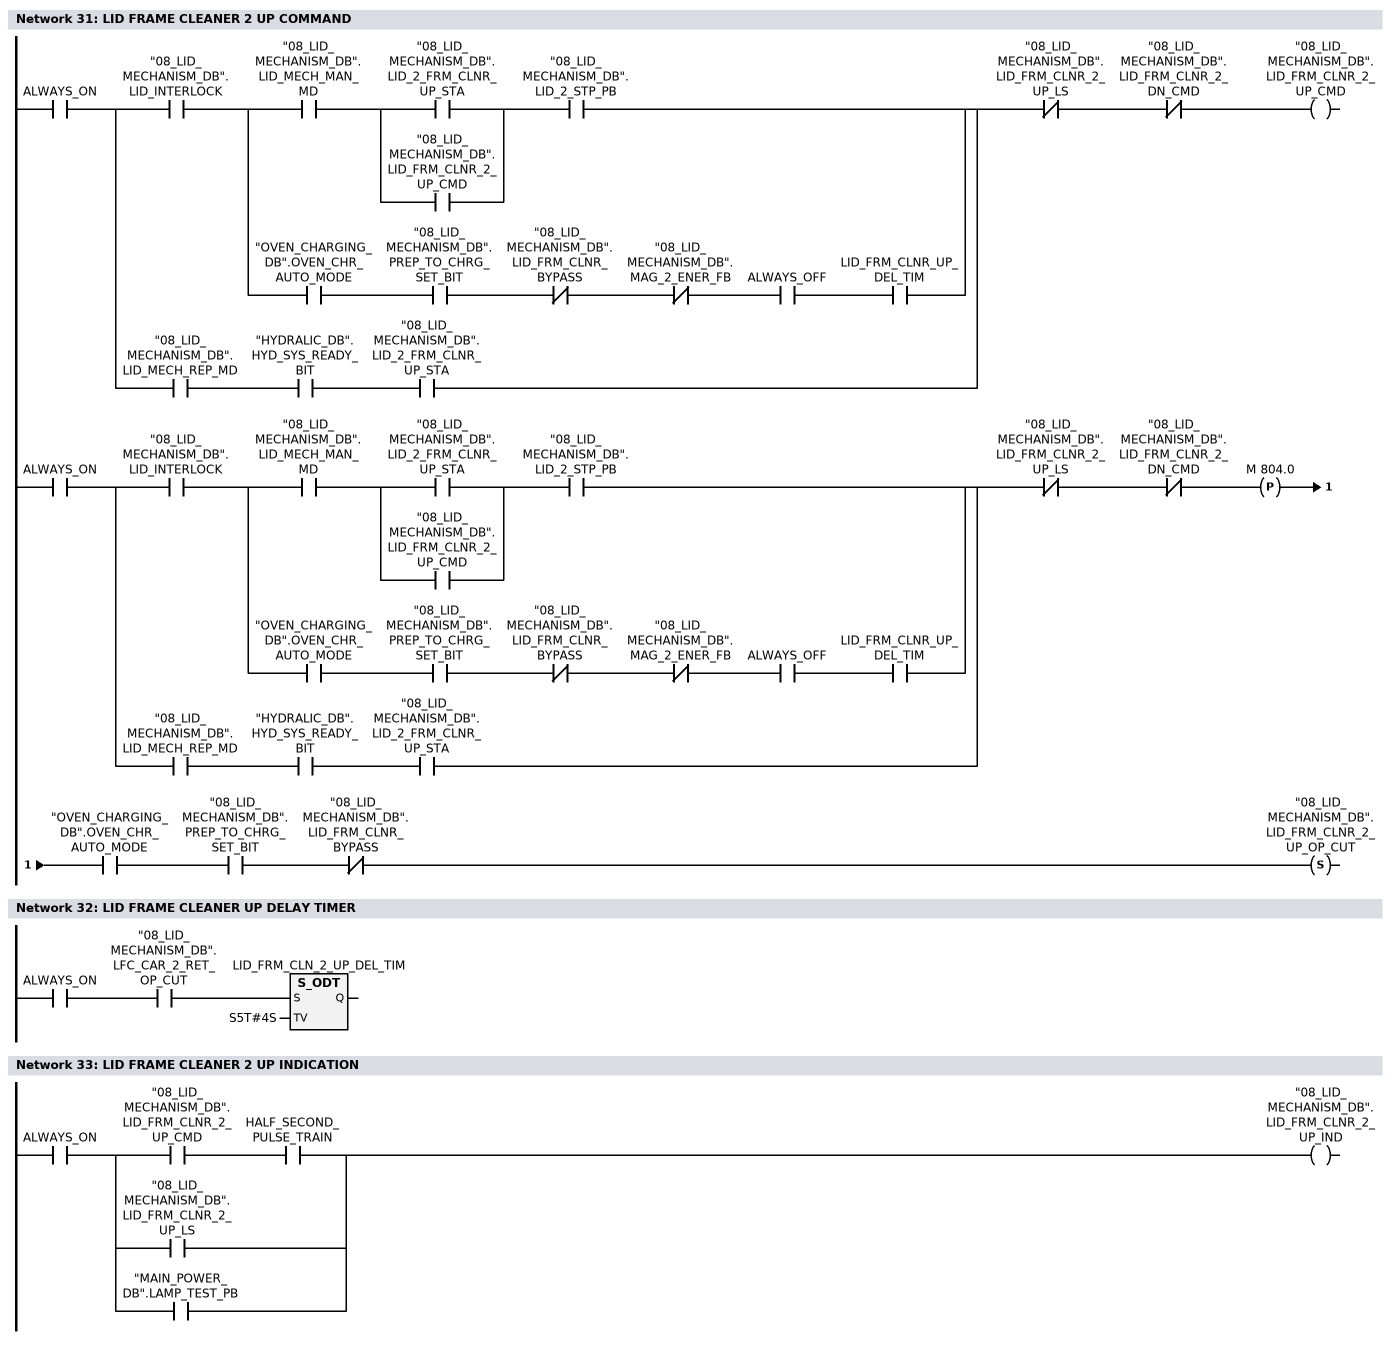
[picture p168: LID_2_MECHANISM networks 31-33]
NETWORK
TITLE = LID FRAME CLEANER 2 UP COMMAND
      A     "ALWAYS_ON";
      A(;
      A     "08_LID_MECHANISM_DB".LID_INTERLOCK;
      A(;
      A     "08_LID_MECHANISM_DB".LID_MECH_MAN_MD;
      A(;
      O     "08_LID_MECHANISM_DB".LID_2_FRM_CLNR_UP_STA;
      O     "08_LID_MECHANISM_DB".LID_FRM_CLNR_2_UP_CMD;
      );
      A     "08_LID_MECHANISM_DB".LID_2_STP_PB;
      O;
      A     "OVEN_CHARGING_DB".OVEN_CHR_AUTO_MODE;
      A     "08_LID_MECHANISM_DB".PREP_TO_CHRG_SET_BIT;
      AN    "08_LID_MECHANISM_DB".LID_FRM_CLNR_BYPASS;
      AN    "08_LID_MECHANISM_DB".MAG_2_ENER_FB;
      A     "ALWAYS_OFF";
      A     "LID_FRM_CLNR_UP_DEL_TIM";
      );
      O;
      A     "08_LID_MECHANISM_DB".LID_MECH_REP_MD;
      A     "HYDRALIC_DB".HYD_SYS_READY_BIT;
      A     "08_LID_MECHANISM_DB".LID_2_FRM_CLNR_UP_STA;
      );
      AN    "08_LID_MECHANISM_DB".LID_FRM_CLNR_2_UP_LS;
      AN    "08_LID_MECHANISM_DB".LID_FRM_CLNR_2_DN_CMD;
      =     L 0.0;
      A     L 0.0;
      BLD   102;
      =     "08_LID_MECHANISM_DB".LID_FRM_CLNR_2_UP_CMD;
      A(;
      A     L 0.0;
      FP    M 804.0;
      );
      A     "OVEN_CHARGING_DB".OVEN_CHR_AUTO_MODE;
      A     "08_LID_MECHANISM_DB".PREP_TO_CHRG_SET_BIT;
      AN    "08_LID_MECHANISM_DB".LID_FRM_CLNR_BYPASS;
      S     "08_LID_MECHANISM_DB".LID_FRM_CLNR_2_UP_OP_CUT;
NETWORK
TITLE = LID FRAME CLEANER UP DELAY TIMER
      A     "ALWAYS_ON";
      A     "08_LID_MECHANISM_DB".LFC_CAR_2_RET_OP_CUT;
      L     S5T#4S;
      SD    "LID_FRM_CLN_2_UP_DEL_TIM";
      NOP   0;
      NOP   0;
      NOP   0;
      NOP   0;
NETWORK
TITLE = LID FRAME CLEANER 2 UP INDICATION
      A     "ALWAYS_ON";
      A(;
      A     "08_LID_MECHANISM_DB".LID_FRM_CLNR_2_UP_CMD;
      A     "HALF_SECOND_PULSE_TRAIN";
      O     "08_LID_MECHANISM_DB".LID_FRM_CLNR_2_UP_LS;
      O     "MAIN_POWER_DB".LAMP_TEST_PB;
      );
      =     "08_LID_MECHANISM_DB".LID_FRM_CLNR_2_UP_IND;
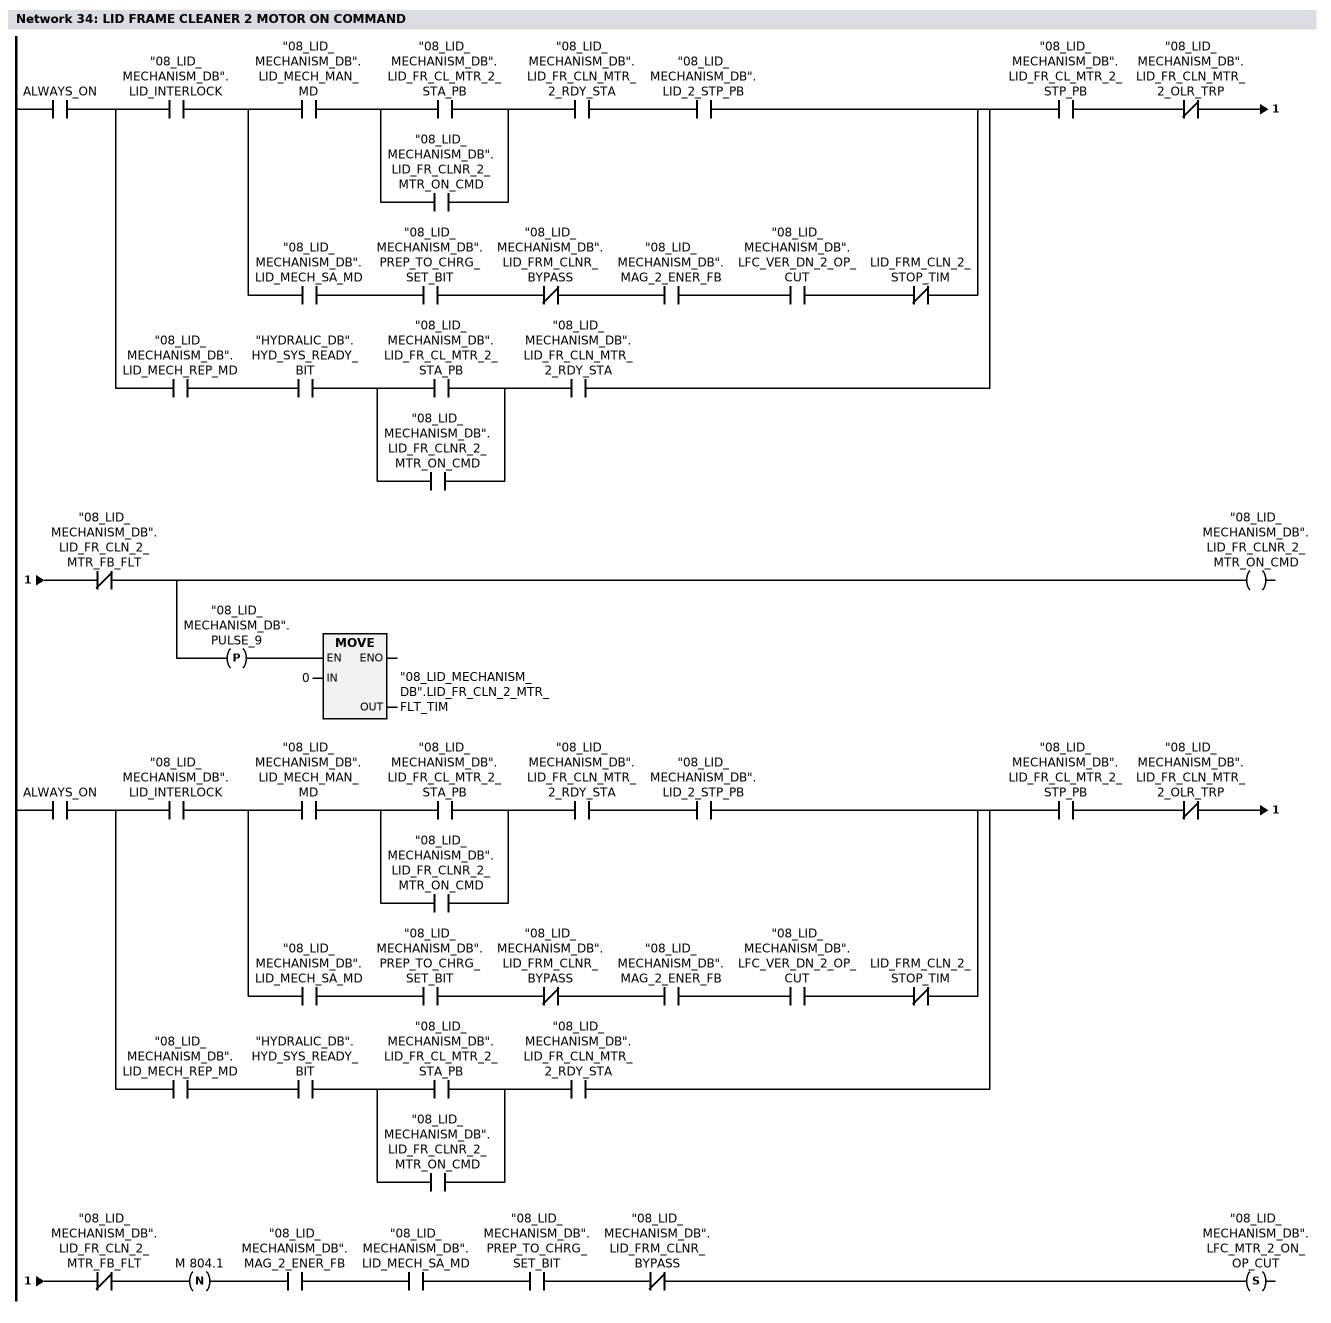
NETWORK
TITLE = LID FRAME CLEANER 2 MOTOR ON COMMAND
      A     "ALWAYS_ON";
      A(;
      A     "08_LID_MECHANISM_DB".LID_INTERLOCK;
      A(;
      A     "08_LID_MECHANISM_DB".LID_MECH_MAN_MD;
      A(;
      O     "08_LID_MECHANISM_DB".LID_FR_CL_MTR_2_STA_PB;
      O     "08_LID_MECHANISM_DB".LID_FR_CLNR_2_MTR_ON_CMD;
      );
      A     "08_LID_MECHANISM_DB".LID_FR_CLN_MTR_2_RDY_STA;
      A     "08_LID_MECHANISM_DB".LID_2_STP_PB;
      O;
      A     "08_LID_MECHANISM_DB".LID_MECH_SA_MD;
      A     "08_LID_MECHANISM_DB".PREP_TO_CHRG_SET_BIT;
      AN    "08_LID_MECHANISM_DB".LID_FRM_CLNR_BYPASS;
      A     "08_LID_MECHANISM_DB".MAG_2_ENER_FB;
      A     "08_LID_MECHANISM_DB".LFC_VER_DN_2_OP_CUT;
      AN    "LID_FRM_CLN_2_STOP_TIM";
      );
      O;
      A     "08_LID_MECHANISM_DB".LID_MECH_REP_MD;
      A     "HYDRALIC_DB".HYD_SYS_READY_BIT;
      A(;
      O     "08_LID_MECHANISM_DB".LID_FR_CL_MTR_2_STA_PB;
      O     "08_LID_MECHANISM_DB".LID_FR_CLNR_2_MTR_ON_CMD;
      );
      A     "08_LID_MECHANISM_DB".LID_FR_CLN_MTR_2_RDY_STA;
      );
      A     "08_LID_MECHANISM_DB".LID_FR_CL_MTR_2_STP_PB;
      AN    "08_LID_MECHANISM_DB".LID_FR_CLN_MTR_2_OLR_TRP;
      AN    "08_LID_MECHANISM_DB".LID_FR_CLN_2_MTR_FB_FLT;
      =     L 0.0;
      A     L 0.0;
      BLD   102;
      =     "08_LID_MECHANISM_DB".LID_FR_CLNR_2_MTR_ON_CMD;
      A     L 0.0;
      FP    "08_LID_MECHANISM_DB".PULSE_9;
      JNB   _00f;
      L     0;
      T     "08_LID_MECHANISM_DB".LID_FR_CLN_2_MTR_FLT_TIM;
_00f: NOP   0;
      A(;
      A     L 0.0;
      FN    M 804.1;
      );
      A     "08_LID_MECHANISM_DB".MAG_2_ENER_FB;
      A     "08_LID_MECHANISM_DB".LID_MECH_SA_MD;
      A     "08_LID_MECHANISM_DB".PREP_TO_CHRG_SET_BIT;
      AN    "08_LID_MECHANISM_DB".LID_FRM_CLNR_BYPASS;
      S     "08_LID_MECHANISM_DB".LFC_MTR_2_ON_OP_CUT;
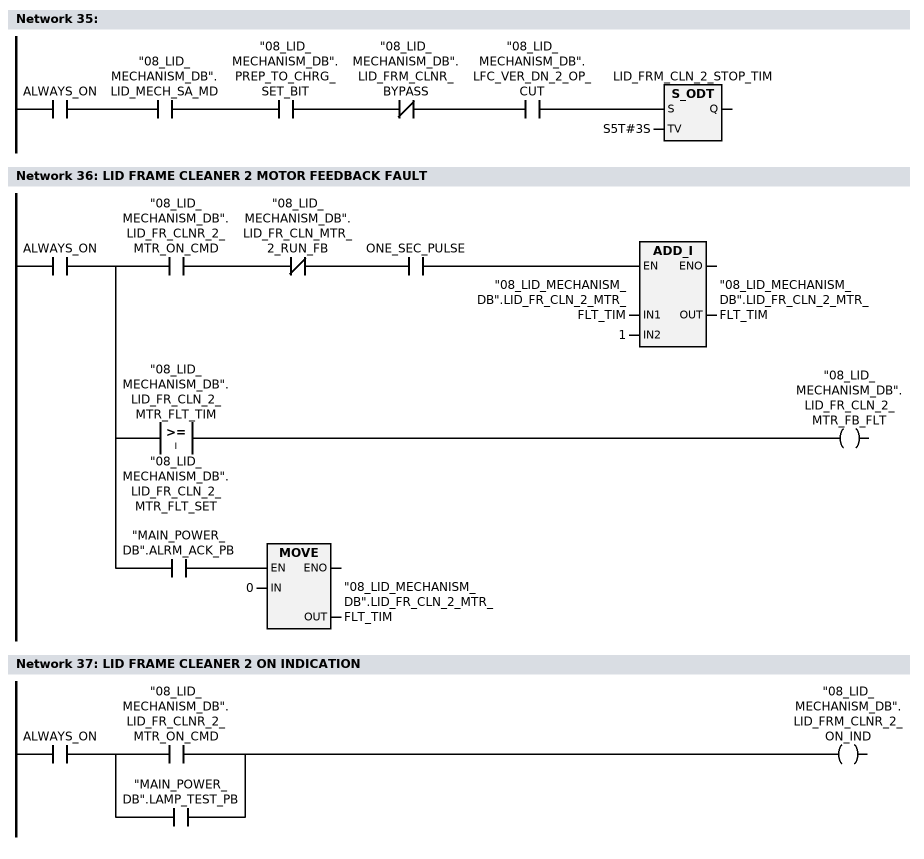
NETWORK
TITLE =
      A     "ALWAYS_ON";
      A     "08_LID_MECHANISM_DB".LID_MECH_SA_MD;
      A     "08_LID_MECHANISM_DB".PREP_TO_CHRG_SET_BIT;
      AN    "08_LID_MECHANISM_DB".LID_FRM_CLNR_BYPASS;
      A     "08_LID_MECHANISM_DB".LFC_VER_DN_2_OP_CUT;
      L     S5T#3S;
      SD    "LID_FRM_CLN_2_STOP_TIM";
      NOP   0;
      NOP   0;
      NOP   0;
      NOP   0;
NETWORK
TITLE = LID FRAME CLEANER 2 MOTOR FEEDBACK FAULT
      A     "ALWAYS_ON";
      =     L 0.0;
      A     L 0.0;
      A     "08_LID_MECHANISM_DB".LID_FR_CLNR_2_MTR_ON_CMD;
      AN    "08_LID_MECHANISM_DB".LID_FR_CLN_MTR_2_RUN_FB;
      A     "ONE_SEC_PULSE";
      JNB   _010;
      L     "08_LID_MECHANISM_DB".LID_FR_CLN_2_MTR_FLT_TIM;
      L     1;
      +I;
      T     "08_LID_MECHANISM_DB".LID_FR_CLN_2_MTR_FLT_TIM;
_010: NOP   0;
      A     L 0.0;
      A(;
      L     "08_LID_MECHANISM_DB".LID_FR_CLN_2_MTR_FLT_TIM;
      L     "08_LID_MECHANISM_DB".LID_FR_CLN_2_MTR_FLT_SET;
      >=I;
      );
      =     "08_LID_MECHANISM_DB".LID_FR_CLN_2_MTR_FB_FLT;
      A     L 0.0;
      A     "MAIN_POWER_DB".ALRM_ACK_PB;
      JNB   _011;
      L     0;
      T     "08_LID_MECHANISM_DB".LID_FR_CLN_2_MTR_FLT_TIM;
_011: NOP   0;
NETWORK
TITLE = LID FRAME CLEANER 2 ON INDICATION
      A     "ALWAYS_ON";
      A(;
      O     "08_LID_MECHANISM_DB".LID_FR_CLNR_2_MTR_ON_CMD;
      O     "MAIN_POWER_DB".LAMP_TEST_PB;
      );
      =     "08_LID_MECHANISM_DB".LID_FRM_CLNR_2_ON_IND;
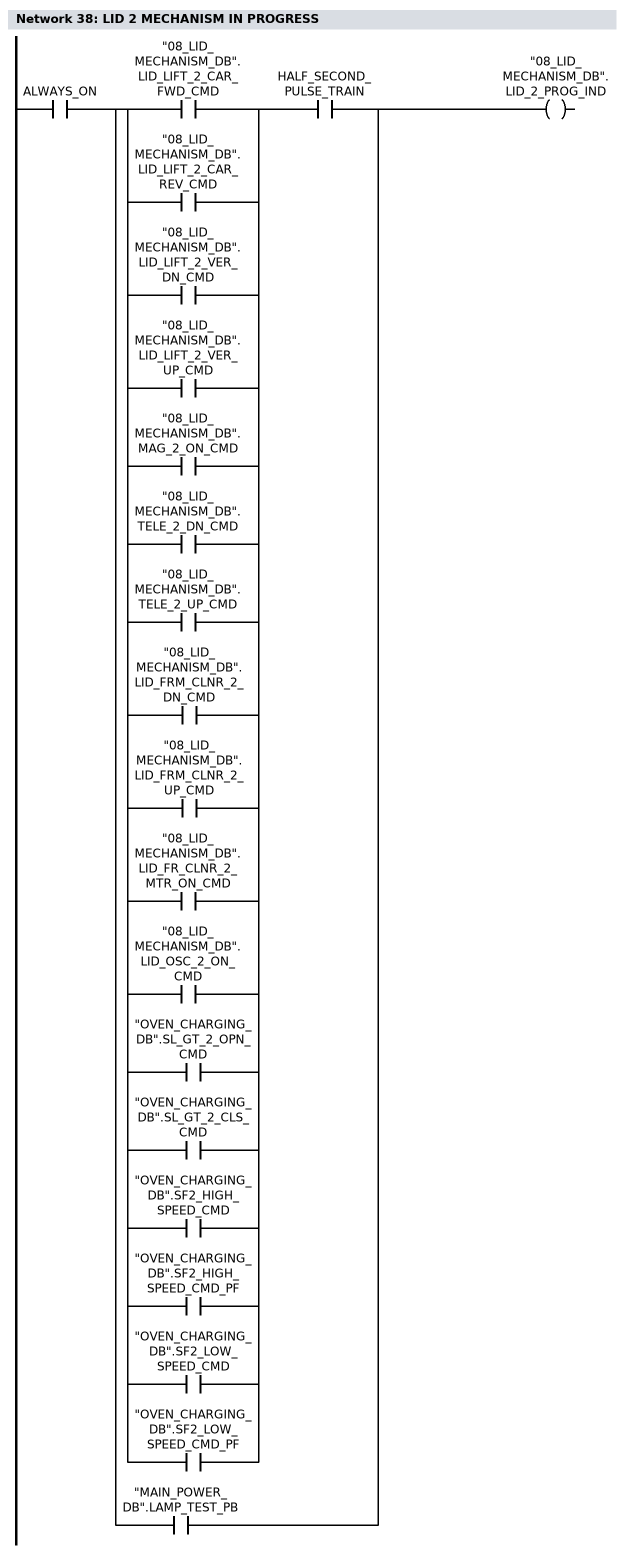
NETWORK
TITLE = LID 2 MECHANISM IN PROGRESS
      A     "ALWAYS_ON";
      A(;
      A(;
      O     "08_LID_MECHANISM_DB".LID_LIFT_2_CAR_FWD_CMD;
      O     "08_LID_MECHANISM_DB".LID_LIFT_2_CAR_REV_CMD;
      O     "08_LID_MECHANISM_DB".LID_LIFT_2_VER_DN_CMD;
      O     "08_LID_MECHANISM_DB".LID_LIFT_2_VER_UP_CMD;
      O     "08_LID_MECHANISM_DB".MAG_2_ON_CMD;
      O     "08_LID_MECHANISM_DB".TELE_2_DN_CMD;
      O     "08_LID_MECHANISM_DB".TELE_2_UP_CMD;
      O     "08_LID_MECHANISM_DB".LID_FRM_CLNR_2_DN_CMD;
      O     "08_LID_MECHANISM_DB".LID_FRM_CLNR_2_UP_CMD;
      O     "08_LID_MECHANISM_DB".LID_FR_CLNR_2_MTR_ON_CMD;
      O     "08_LID_MECHANISM_DB".LID_OSC_2_ON_CMD;
      O     "OVEN_CHARGING_DB".SL_GT_2_OPN_CMD;
      O     "OVEN_CHARGING_DB".SL_GT_2_CLS_CMD;
      O     "OVEN_CHARGING_DB".SF2_HIGH_SPEED_CMD;
      O     "OVEN_CHARGING_DB".SF2_HIGH_SPEED_CMD_PF;
      O     "OVEN_CHARGING_DB".SF2_LOW_SPEED_CMD;
      O     "OVEN_CHARGING_DB".SF2_LOW_SPEED_CMD_PF;
      );
      A     "HALF_SECOND_PULSE_TRAIN";
      O     "MAIN_POWER_DB".LAMP_TEST_PB;
      );
      =     "08_LID_MECHANISM_DB".LID_2_PROG_IND;
END_FUNCTION

FUNCTION "LID_3_MECHANISM" : VOID	// FC 14
//AUTO SEQ
//Prepare to charge pb 
//Carriage Fwd 
//Vert Down 
//Mag On
//Osc On
//3s 
//Osc off
//Lid at mag
//Ver Up
//Car Ret 
//// Frm clnr down if bypass
//Car fwd 
//car Ver cln pos down 
//Frm clnr Mtr on 
//5s 
//off 
//car Ver  up 
//Car Ret //
//Teles Down 
AUTHOR : Arun
VERSION : 0.1
BEGIN
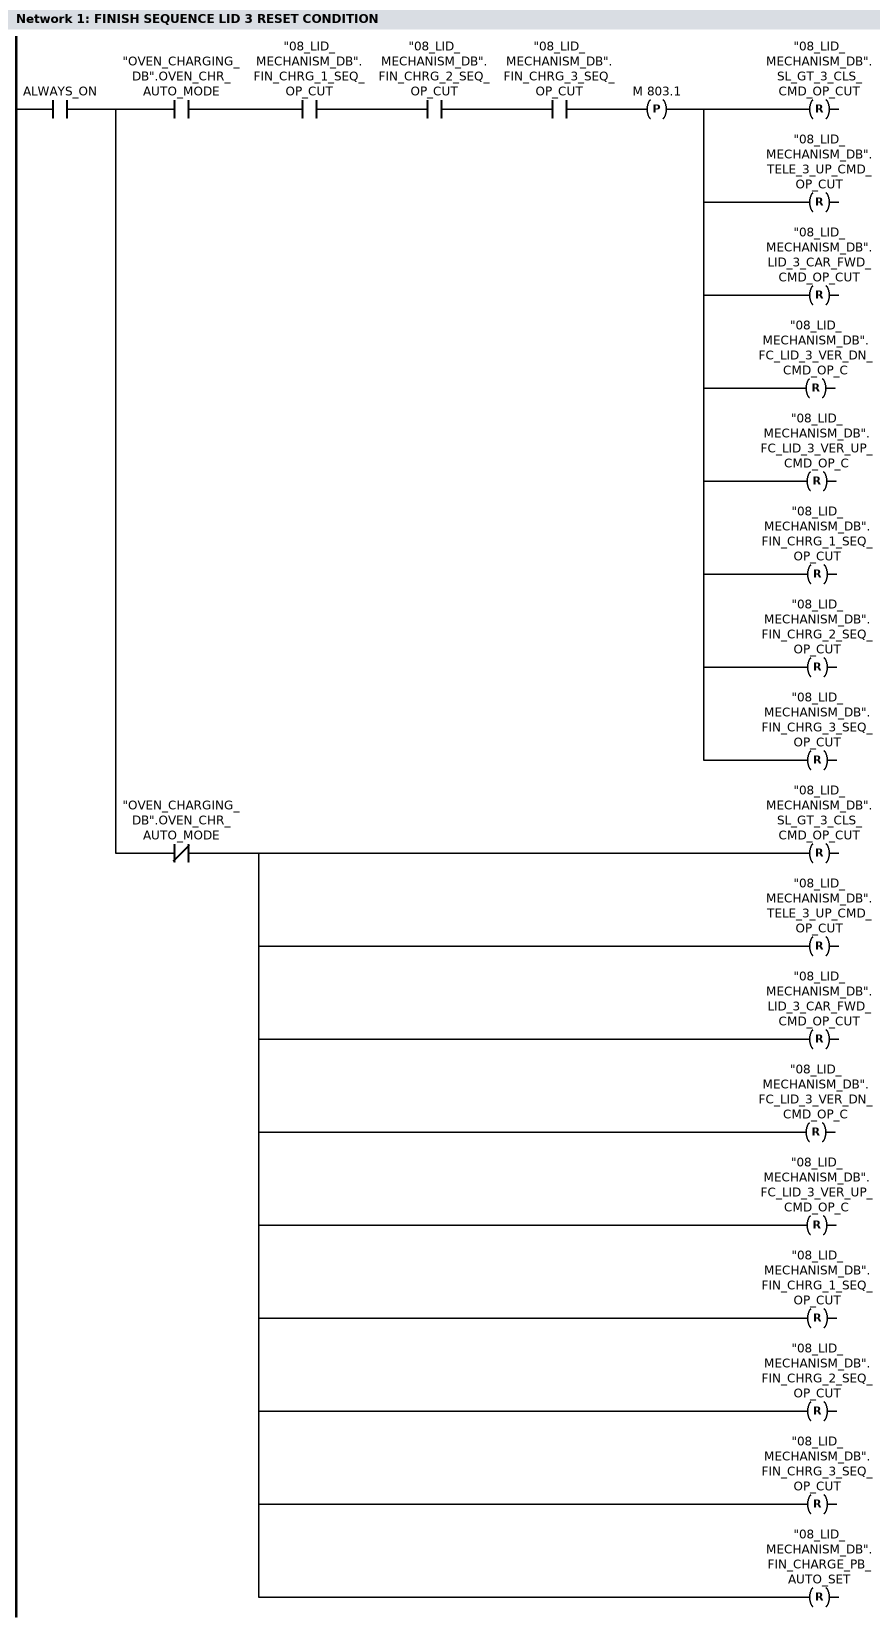
NETWORK
TITLE = FINISH SEQUENCE LID 3 RESET CONDITION
      A     "ALWAYS_ON";
      =     L 0.0;
      A     L 0.0;
      A     "OVEN_CHARGING_DB".OVEN_CHR_AUTO_MODE;
      A     "08_LID_MECHANISM_DB".FIN_CHRG_1_SEQ_OP_CUT;
      A     "08_LID_MECHANISM_DB".FIN_CHRG_2_SEQ_OP_CUT;
      A     "08_LID_MECHANISM_DB".FIN_CHRG_3_SEQ_OP_CUT;
      FP    M 803.1;
      R     "08_LID_MECHANISM_DB".SL_GT_3_CLS_CMD_OP_CUT;
      R     "08_LID_MECHANISM_DB".TELE_3_UP_CMD_OP_CUT;
      R     "08_LID_MECHANISM_DB".LID_3_CAR_FWD_CMD_OP_CUT;
      R     "08_LID_MECHANISM_DB".FC_LID_3_VER_DN_CMD_OP_C;
      R     "08_LID_MECHANISM_DB".FC_LID_3_VER_UP_CMD_OP_C;
      R     "08_LID_MECHANISM_DB".FIN_CHRG_1_SEQ_OP_CUT;
      R     "08_LID_MECHANISM_DB".FIN_CHRG_2_SEQ_OP_CUT;
      R     "08_LID_MECHANISM_DB".FIN_CHRG_3_SEQ_OP_CUT;
      A     L 0.0;
      AN    "OVEN_CHARGING_DB".OVEN_CHR_AUTO_MODE;
      R     "08_LID_MECHANISM_DB".SL_GT_3_CLS_CMD_OP_CUT;
      R     "08_LID_MECHANISM_DB".TELE_3_UP_CMD_OP_CUT;
      R     "08_LID_MECHANISM_DB".LID_3_CAR_FWD_CMD_OP_CUT;
      R     "08_LID_MECHANISM_DB".FC_LID_3_VER_DN_CMD_OP_C;
      R     "08_LID_MECHANISM_DB".FC_LID_3_VER_UP_CMD_OP_C;
      R     "08_LID_MECHANISM_DB".FIN_CHRG_1_SEQ_OP_CUT;
      R     "08_LID_MECHANISM_DB".FIN_CHRG_2_SEQ_OP_CUT;
      R     "08_LID_MECHANISM_DB".FIN_CHRG_3_SEQ_OP_CUT;
      R     "08_LID_MECHANISM_DB".FIN_CHARGE_PB_AUTO_SET;
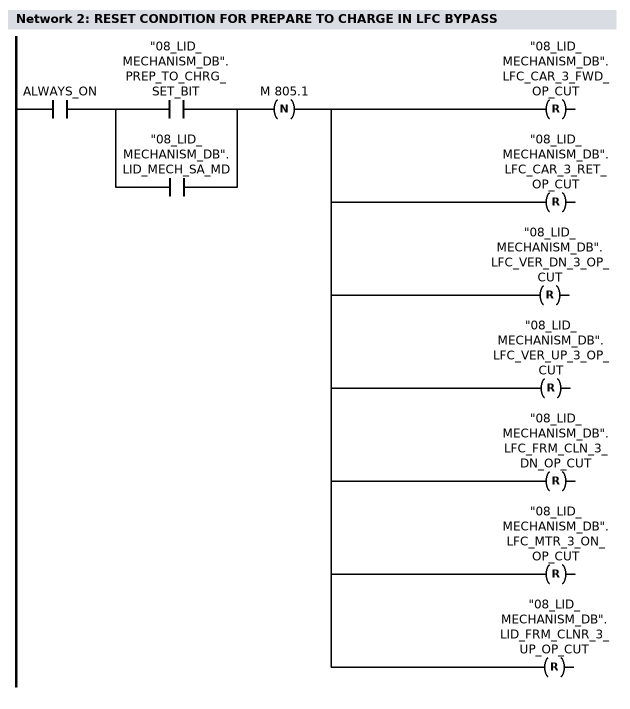
NETWORK
TITLE = RESET CONDITION FOR PREPARE TO CHARGE IN LFC BYPASS
      A     "ALWAYS_ON";
      A(;
      O     "08_LID_MECHANISM_DB".PREP_TO_CHRG_SET_BIT;
      O     "08_LID_MECHANISM_DB".LID_MECH_SA_MD;
      );
      FN    M 805.1;
      R     "08_LID_MECHANISM_DB".LFC_CAR_3_FWD_OP_CUT;
      R     "08_LID_MECHANISM_DB".LFC_CAR_3_RET_OP_CUT;
      R     "08_LID_MECHANISM_DB".LFC_VER_DN_3_OP_CUT;
      R     "08_LID_MECHANISM_DB".LFC_VER_UP_3_OP_CUT;
      R     "08_LID_MECHANISM_DB".LFC_FRM_CLN_3_DN_OP_CUT;
      R     "08_LID_MECHANISM_DB".LFC_MTR_3_ON_OP_CUT;
      R     "08_LID_MECHANISM_DB".LID_FRM_CLNR_3_UP_OP_CUT;
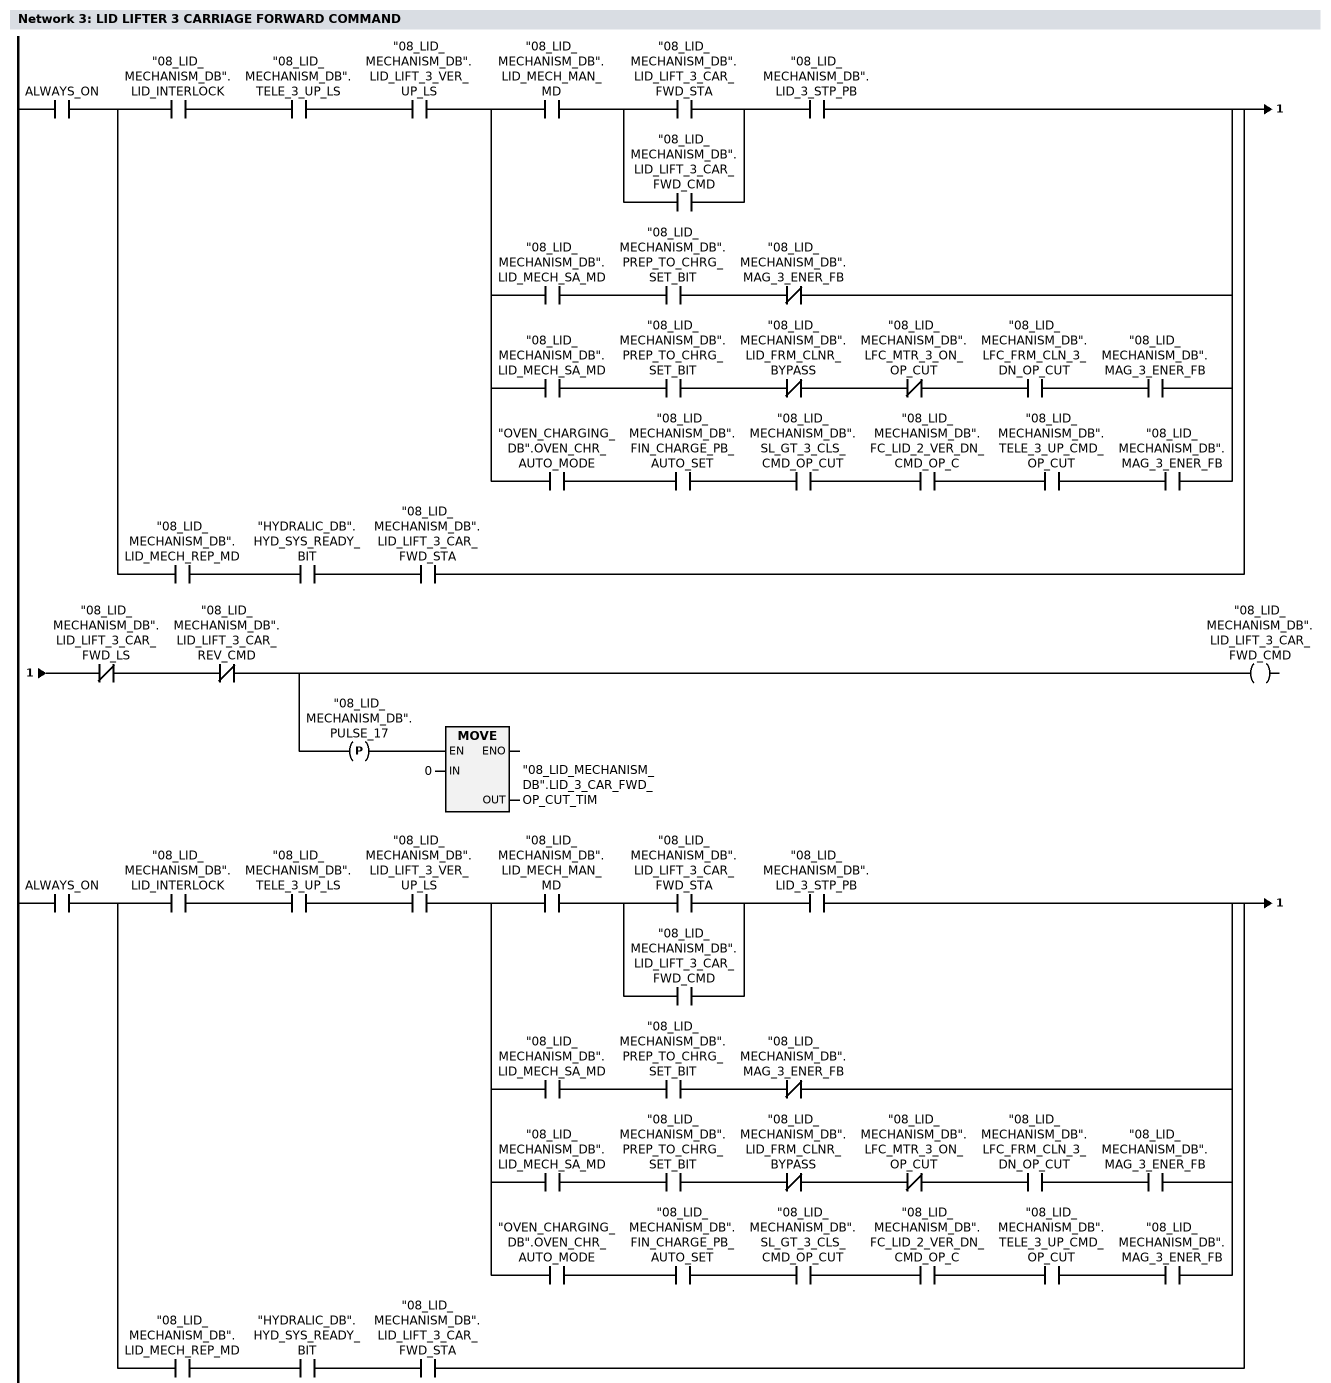
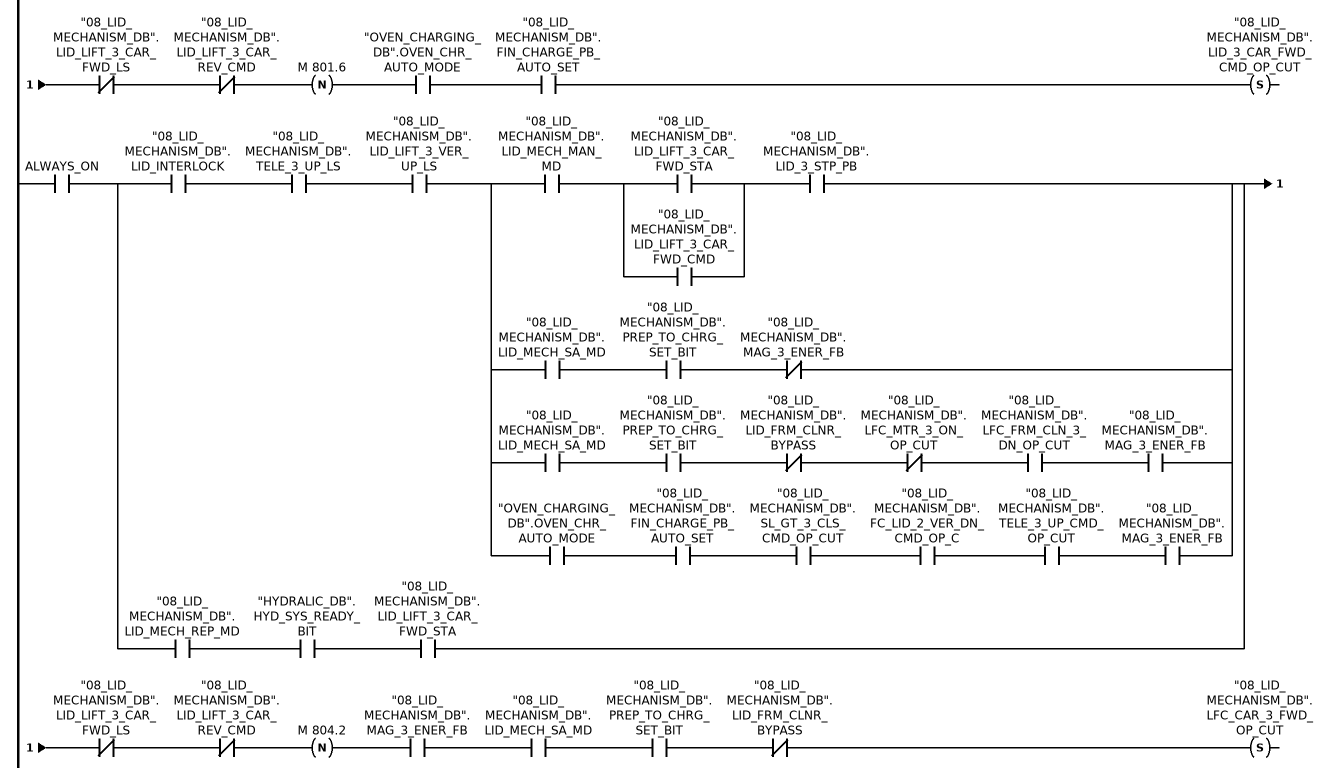
NETWORK
TITLE = LID LIFTER 3 CARRIAGE FORWARD COMMAND
      A     "ALWAYS_ON";
      A(;
      A     "08_LID_MECHANISM_DB".LID_INTERLOCK;
      A     "08_LID_MECHANISM_DB".TELE_3_UP_LS;
      A     "08_LID_MECHANISM_DB".LID_LIFT_3_VER_UP_LS;
      A(;
      A     "08_LID_MECHANISM_DB".LID_MECH_MAN_MD;
      A(;
      O     "08_LID_MECHANISM_DB".LID_LIFT_3_CAR_FWD_STA;
      O     "08_LID_MECHANISM_DB".LID_LIFT_3_CAR_FWD_CMD;
      );
      A     "08_LID_MECHANISM_DB".LID_3_STP_PB;
      O;
      A     "08_LID_MECHANISM_DB".LID_MECH_SA_MD;
      A     "08_LID_MECHANISM_DB".PREP_TO_CHRG_SET_BIT;
      AN    "08_LID_MECHANISM_DB".MAG_3_ENER_FB;
      O;
      A     "08_LID_MECHANISM_DB".LID_MECH_SA_MD;
      A     "08_LID_MECHANISM_DB".PREP_TO_CHRG_SET_BIT;
      AN    "08_LID_MECHANISM_DB".LID_FRM_CLNR_BYPASS;
      AN    "08_LID_MECHANISM_DB".LFC_MTR_3_ON_OP_CUT;
      A     "08_LID_MECHANISM_DB".LFC_FRM_CLN_3_DN_OP_CUT;
      A     "08_LID_MECHANISM_DB".MAG_3_ENER_FB;
      O;
      A     "OVEN_CHARGING_DB".OVEN_CHR_AUTO_MODE;
      A     "08_LID_MECHANISM_DB".FIN_CHARGE_PB_AUTO_SET;
      A     "08_LID_MECHANISM_DB".SL_GT_3_CLS_CMD_OP_CUT;
      A     "08_LID_MECHANISM_DB".FC_LID_2_VER_DN_CMD_OP_C;
      A     "08_LID_MECHANISM_DB".TELE_3_UP_CMD_OP_CUT;
      A     "08_LID_MECHANISM_DB".MAG_3_ENER_FB;
      );
      O;
      A     "08_LID_MECHANISM_DB".LID_MECH_REP_MD;
      A     "HYDRALIC_DB".HYD_SYS_READY_BIT;
      A     "08_LID_MECHANISM_DB".LID_LIFT_3_CAR_FWD_STA;
      );
      AN    "08_LID_MECHANISM_DB".LID_LIFT_3_CAR_FWD_LS;
      AN    "08_LID_MECHANISM_DB".LID_LIFT_3_CAR_REV_CMD;
      =     L 0.0;
      A     L 0.0;
      BLD   102;
      =     "08_LID_MECHANISM_DB".LID_LIFT_3_CAR_FWD_CMD;
      A     L 0.0;
      FP    "08_LID_MECHANISM_DB".PULSE_17;
      JNB   _001;
      L     0;
      T     "08_LID_MECHANISM_DB".LID_3_CAR_FWD_OP_CUT_TIM;
_001: NOP   0;
      A(;
      A     L 0.0;
      FN    M 801.6;
      );
      A     "OVEN_CHARGING_DB".OVEN_CHR_AUTO_MODE;
      A     "08_LID_MECHANISM_DB".FIN_CHARGE_PB_AUTO_SET;
      S     "08_LID_MECHANISM_DB".LID_3_CAR_FWD_CMD_OP_CUT;
      A(;
      A     L 0.0;
      FN    M 804.2;
      );
      A     "08_LID_MECHANISM_DB".MAG_3_ENER_FB;
      A     "08_LID_MECHANISM_DB".LID_MECH_SA_MD;
      A     "08_LID_MECHANISM_DB".PREP_TO_CHRG_SET_BIT;
      AN    "08_LID_MECHANISM_DB".LID_FRM_CLNR_BYPASS;
      S     "08_LID_MECHANISM_DB".LFC_CAR_3_FWD_OP_CUT;
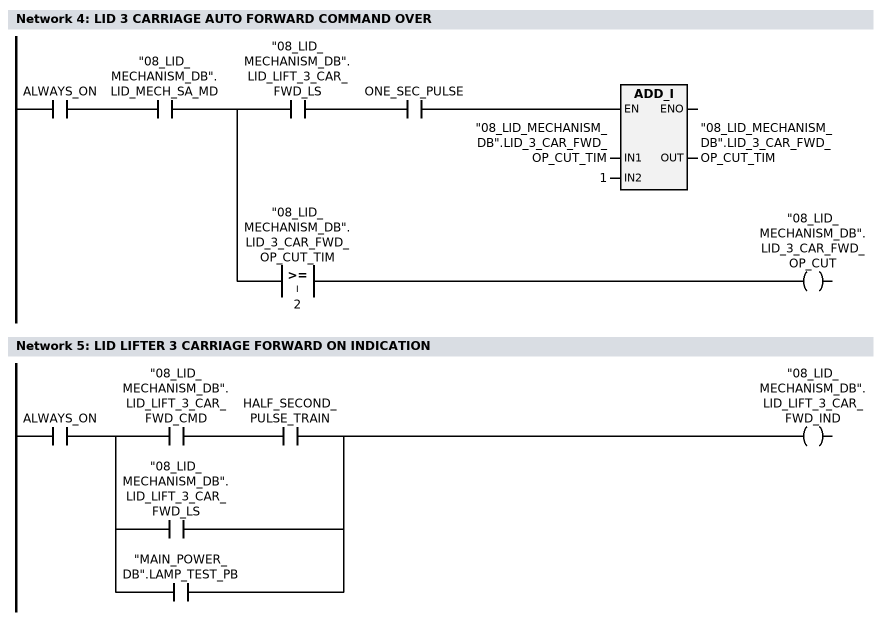
NETWORK
TITLE = LID 3 CARRIAGE AUTO FORWARD COMMAND OVER
      A     "ALWAYS_ON";
      A     "08_LID_MECHANISM_DB".LID_MECH_SA_MD;
      =     L 0.0;
      A     L 0.0;
      A     "08_LID_MECHANISM_DB".LID_LIFT_3_CAR_FWD_LS;
      A     "ONE_SEC_PULSE";
      JNB   _002;
      L     "08_LID_MECHANISM_DB".LID_3_CAR_FWD_OP_CUT_TIM;
      L     1;
      +I;
      T     "08_LID_MECHANISM_DB".LID_3_CAR_FWD_OP_CUT_TIM;
_002: NOP   0;
      A     L 0.0;
      A(;
      L     "08_LID_MECHANISM_DB".LID_3_CAR_FWD_OP_CUT_TIM;
      L     2;
      >=I;
      );
      =     "08_LID_MECHANISM_DB".LID_3_CAR_FWD_OP_CUT;
NETWORK
TITLE = LID LIFTER 3 CARRIAGE FORWARD ON INDICATION
      A     "ALWAYS_ON";
      A(;
      A     "08_LID_MECHANISM_DB".LID_LIFT_3_CAR_FWD_CMD;
      A     "HALF_SECOND_PULSE_TRAIN";
      O     "08_LID_MECHANISM_DB".LID_LIFT_3_CAR_FWD_LS;
      O     "MAIN_POWER_DB".LAMP_TEST_PB;
      );
      =     "08_LID_MECHANISM_DB".LID_LIFT_3_CAR_FWD_IND;
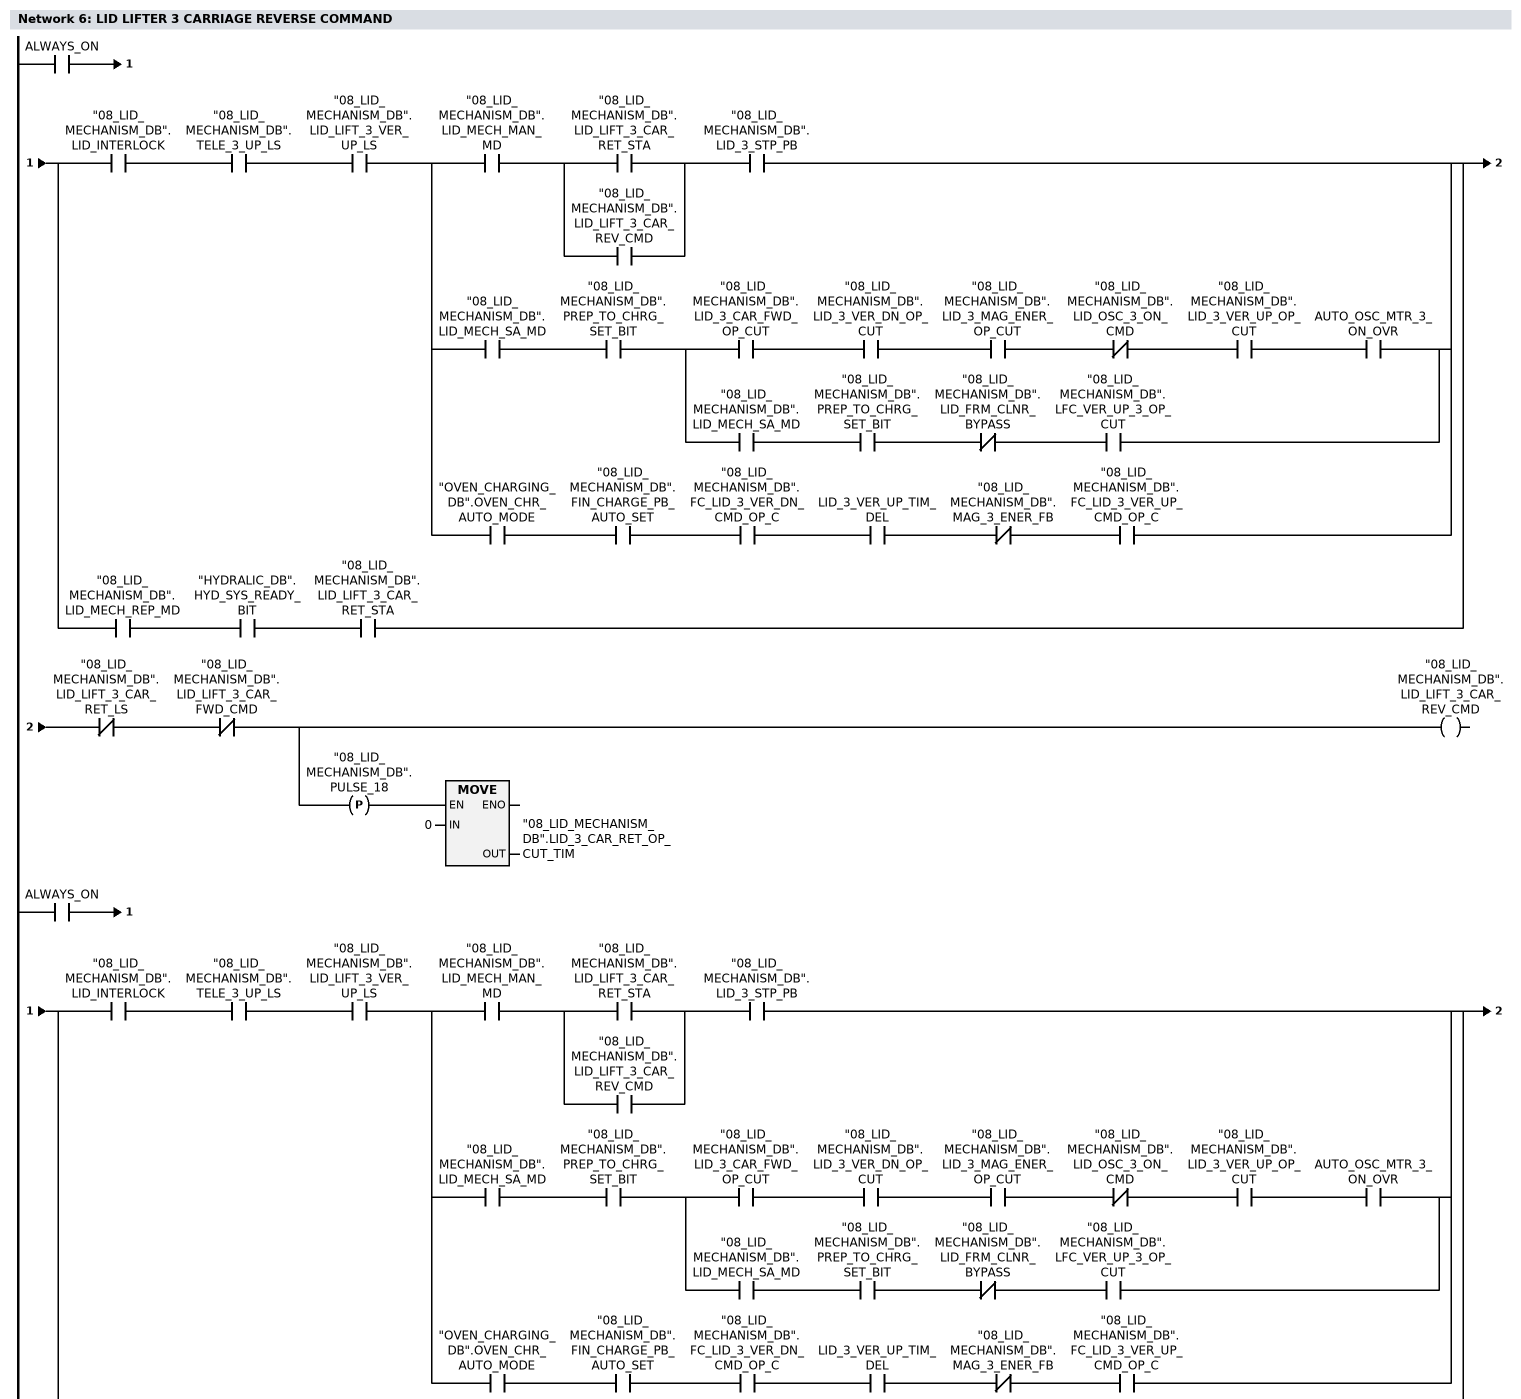
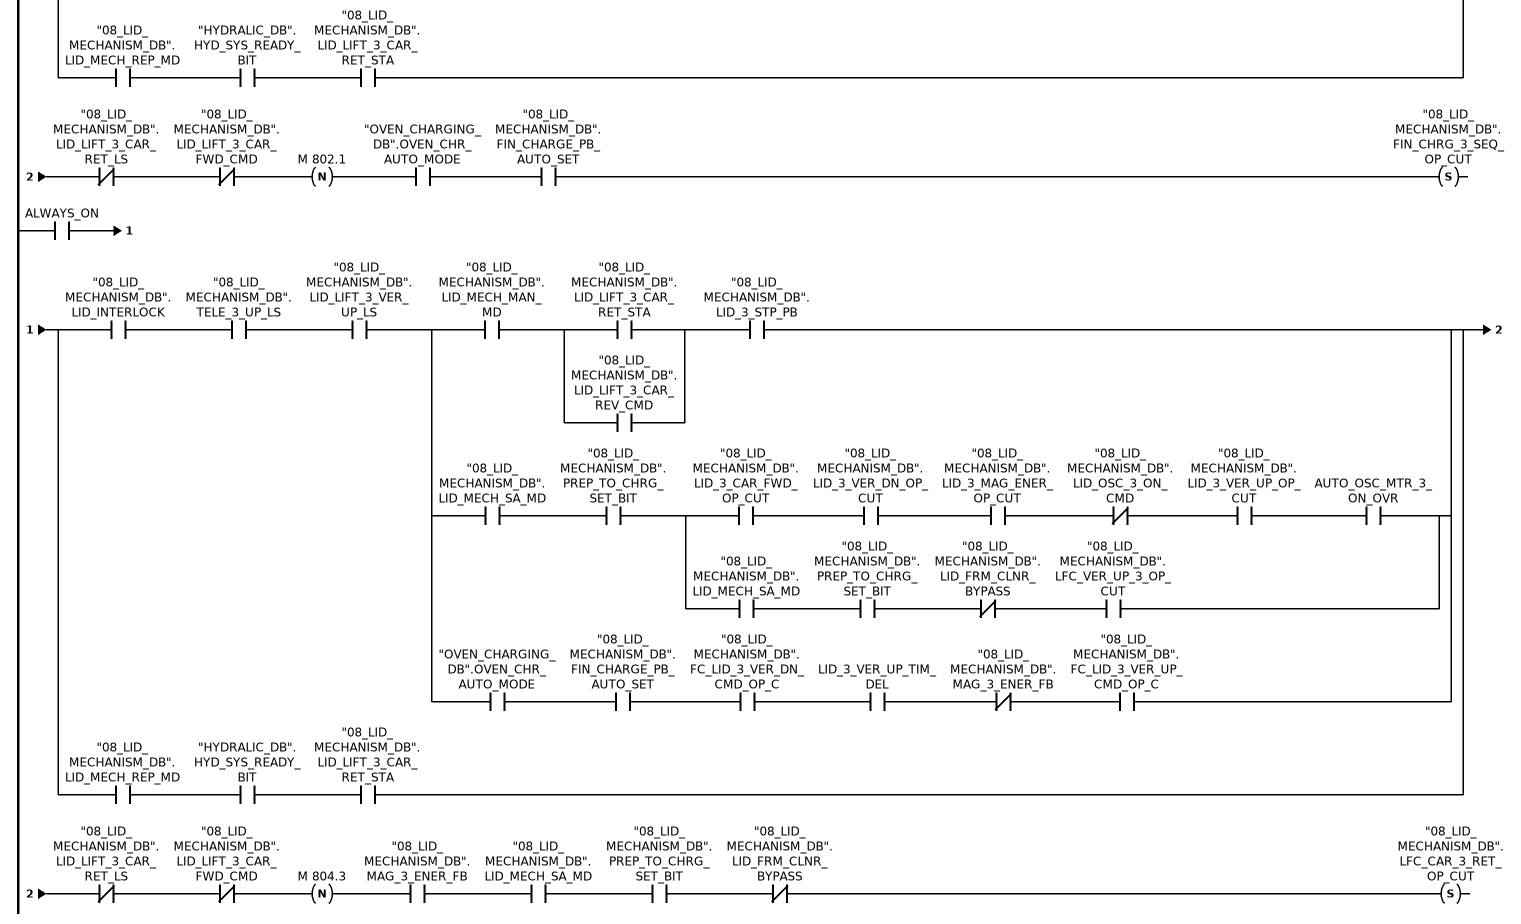
NETWORK
TITLE = LID LIFTER 3 CARRIAGE REVERSE COMMAND
      A     "ALWAYS_ON";
      A(;
      A     "08_LID_MECHANISM_DB".LID_INTERLOCK;
      A     "08_LID_MECHANISM_DB".TELE_3_UP_LS;
      A     "08_LID_MECHANISM_DB".LID_LIFT_3_VER_UP_LS;
      A(;
      A     "08_LID_MECHANISM_DB".LID_MECH_MAN_MD;
      A(;
      O     "08_LID_MECHANISM_DB".LID_LIFT_3_CAR_RET_STA;
      O     "08_LID_MECHANISM_DB".LID_LIFT_3_CAR_REV_CMD;
      );
      A     "08_LID_MECHANISM_DB".LID_3_STP_PB;
      O;
      A     "08_LID_MECHANISM_DB".LID_MECH_SA_MD;
      A     "08_LID_MECHANISM_DB".PREP_TO_CHRG_SET_BIT;
      A(;
      A     "08_LID_MECHANISM_DB".LID_3_CAR_FWD_OP_CUT;
      A     "08_LID_MECHANISM_DB".LID_3_VER_DN_OP_CUT;
      A     "08_LID_MECHANISM_DB".LID_3_MAG_ENER_OP_CUT;
      AN    "08_LID_MECHANISM_DB".LID_OSC_3_ON_CMD;
      A     "08_LID_MECHANISM_DB".LID_3_VER_UP_OP_CUT;
      A     "AUTO_OSC_MTR_3_ON_OVR";
      O;
      A     "08_LID_MECHANISM_DB".LID_MECH_SA_MD;
      A     "08_LID_MECHANISM_DB".PREP_TO_CHRG_SET_BIT;
      AN    "08_LID_MECHANISM_DB".LID_FRM_CLNR_BYPASS;
      A     "08_LID_MECHANISM_DB".LFC_VER_UP_3_OP_CUT;
      );
      O;
      A     "OVEN_CHARGING_DB".OVEN_CHR_AUTO_MODE;
      A     "08_LID_MECHANISM_DB".FIN_CHARGE_PB_AUTO_SET;
      A     "08_LID_MECHANISM_DB".FC_LID_3_VER_DN_CMD_OP_C;
      A     "LID_3_VER_UP_TIM_DEL";
      AN    "08_LID_MECHANISM_DB".MAG_3_ENER_FB;
      A     "08_LID_MECHANISM_DB".FC_LID_3_VER_UP_CMD_OP_C;
      );
      O;
      A     "08_LID_MECHANISM_DB".LID_MECH_REP_MD;
      A     "HYDRALIC_DB".HYD_SYS_READY_BIT;
      A     "08_LID_MECHANISM_DB".LID_LIFT_3_CAR_RET_STA;
      );
      AN    "08_LID_MECHANISM_DB".LID_LIFT_3_CAR_RET_LS;
      AN    "08_LID_MECHANISM_DB".LID_LIFT_3_CAR_FWD_CMD;
      =     L 0.0;
      A     L 0.0;
      BLD   102;
      =     "08_LID_MECHANISM_DB".LID_LIFT_3_CAR_REV_CMD;
      A     L 0.0;
      FP    "08_LID_MECHANISM_DB".PULSE_18;
      JNB   _003;
      L     0;
      T     "08_LID_MECHANISM_DB".LID_3_CAR_RET_OP_CUT_TIM;
_003: NOP   0;
      A(;
      A     L 0.0;
      FN    M 802.1;
      );
      A     "OVEN_CHARGING_DB".OVEN_CHR_AUTO_MODE;
      A     "08_LID_MECHANISM_DB".FIN_CHARGE_PB_AUTO_SET;
      S     "08_LID_MECHANISM_DB".FIN_CHRG_3_SEQ_OP_CUT;
      A(;
      A     L 0.0;
      FN    M 804.3;
      );
      A     "08_LID_MECHANISM_DB".MAG_3_ENER_FB;
      A     "08_LID_MECHANISM_DB".LID_MECH_SA_MD;
      A     "08_LID_MECHANISM_DB".PREP_TO_CHRG_SET_BIT;
      AN    "08_LID_MECHANISM_DB".LID_FRM_CLNR_BYPASS;
      S     "08_LID_MECHANISM_DB".LFC_CAR_3_RET_OP_CUT;
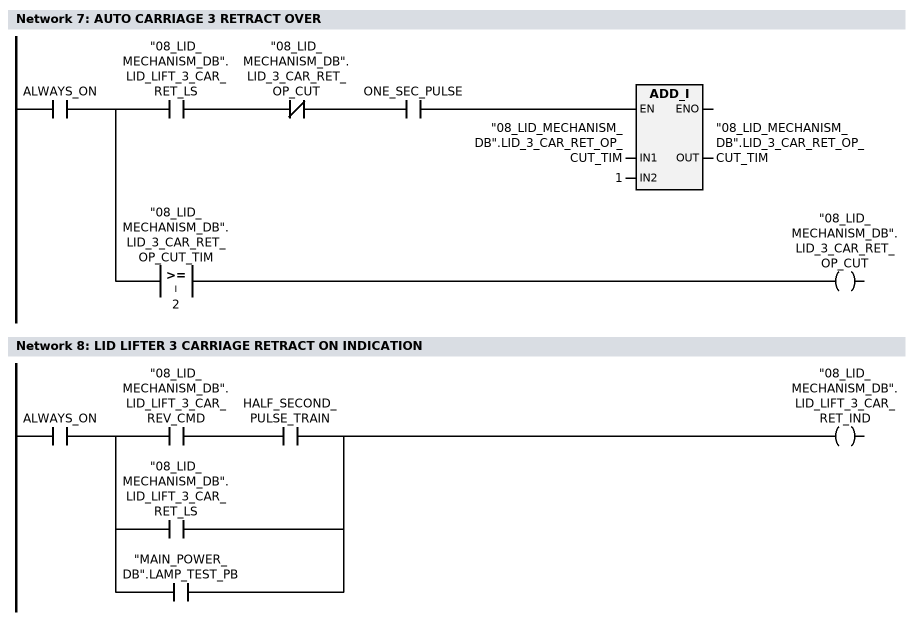
NETWORK
TITLE = AUTO CARRIAGE 3 RETRACT OVER
      A     "ALWAYS_ON";
      =     L 0.0;
      A     L 0.0;
      A     "08_LID_MECHANISM_DB".LID_LIFT_3_CAR_RET_LS;
      AN    "08_LID_MECHANISM_DB".LID_3_CAR_RET_OP_CUT;
      A     "ONE_SEC_PULSE";
      JNB   _004;
      L     "08_LID_MECHANISM_DB".LID_3_CAR_RET_OP_CUT_TIM;
      L     1;
      +I;
      T     "08_LID_MECHANISM_DB".LID_3_CAR_RET_OP_CUT_TIM;
_004: NOP   0;
      A     L 0.0;
      A(;
      L     "08_LID_MECHANISM_DB".LID_3_CAR_RET_OP_CUT_TIM;
      L     2;
      >=I;
      );
      =     "08_LID_MECHANISM_DB".LID_3_CAR_RET_OP_CUT;
NETWORK
TITLE = LID LIFTER 3 CARRIAGE RETRACT ON INDICATION
      A     "ALWAYS_ON";
      A(;
      A     "08_LID_MECHANISM_DB".LID_LIFT_3_CAR_REV_CMD;
      A     "HALF_SECOND_PULSE_TRAIN";
      O     "08_LID_MECHANISM_DB".LID_LIFT_3_CAR_RET_LS;
      O     "MAIN_POWER_DB".LAMP_TEST_PB;
      );
      =     "08_LID_MECHANISM_DB".LID_LIFT_3_CAR_RET_IND;
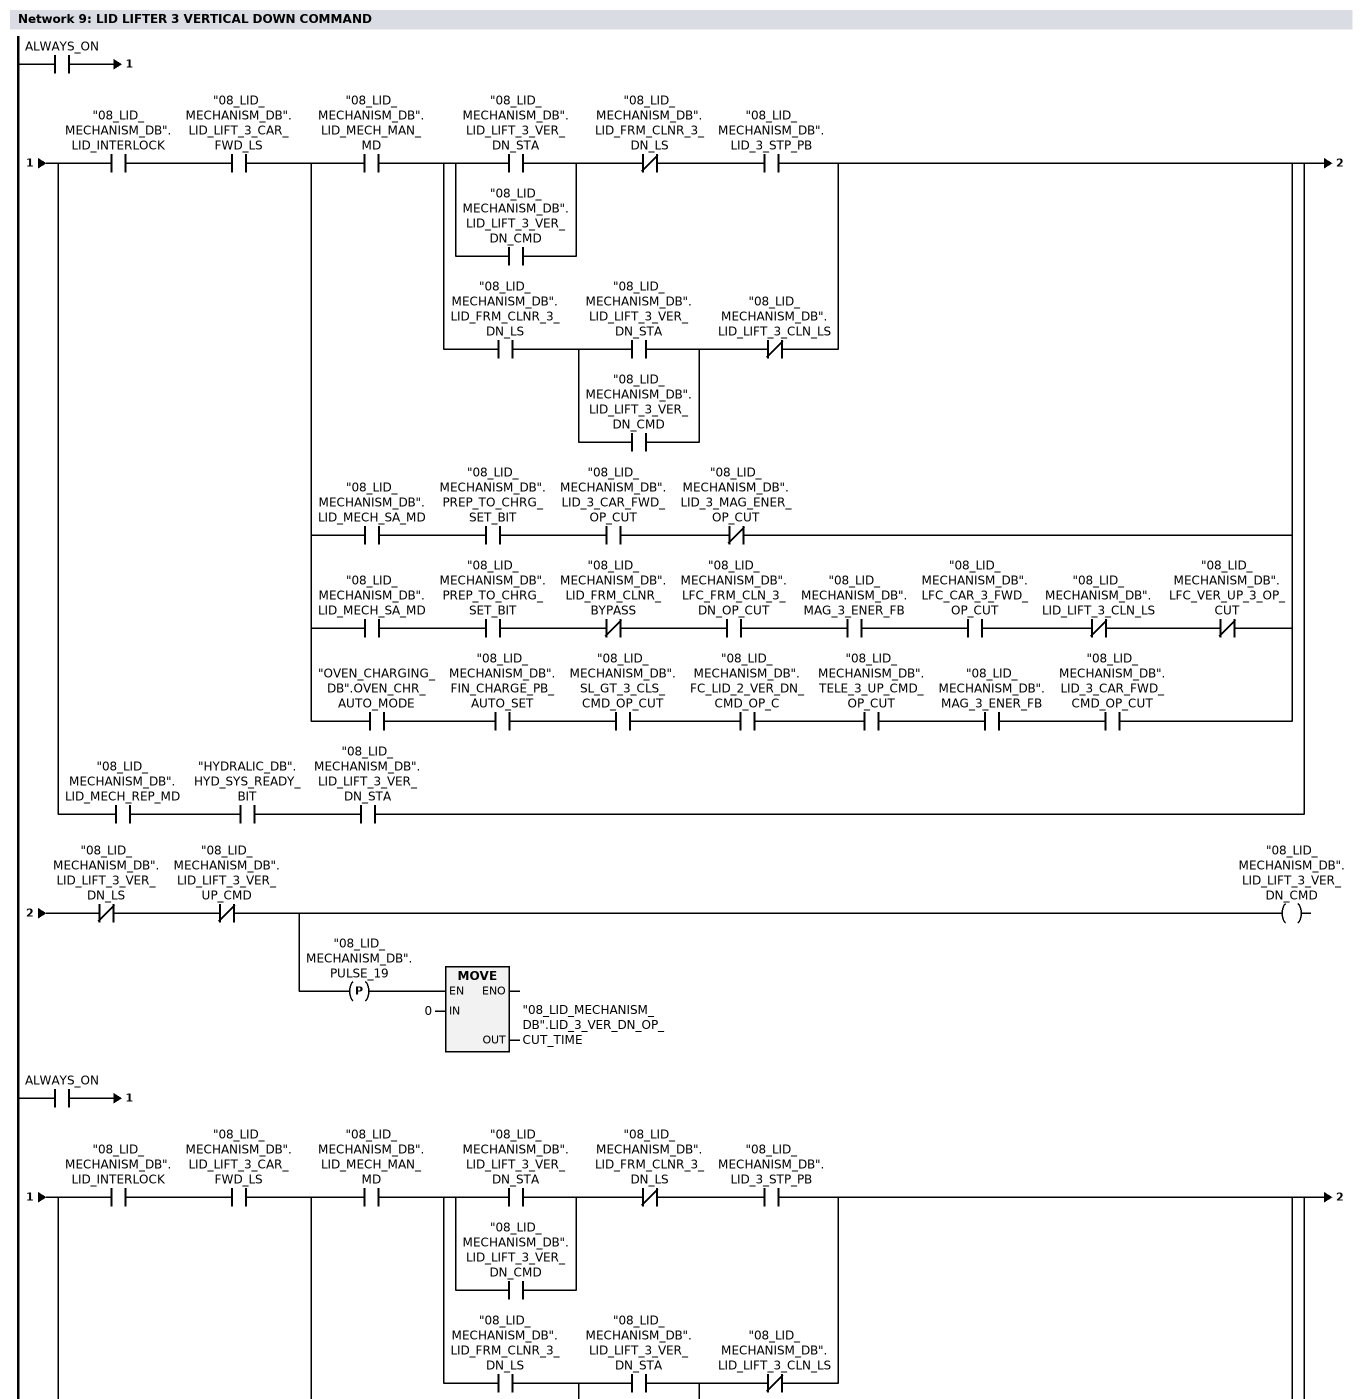
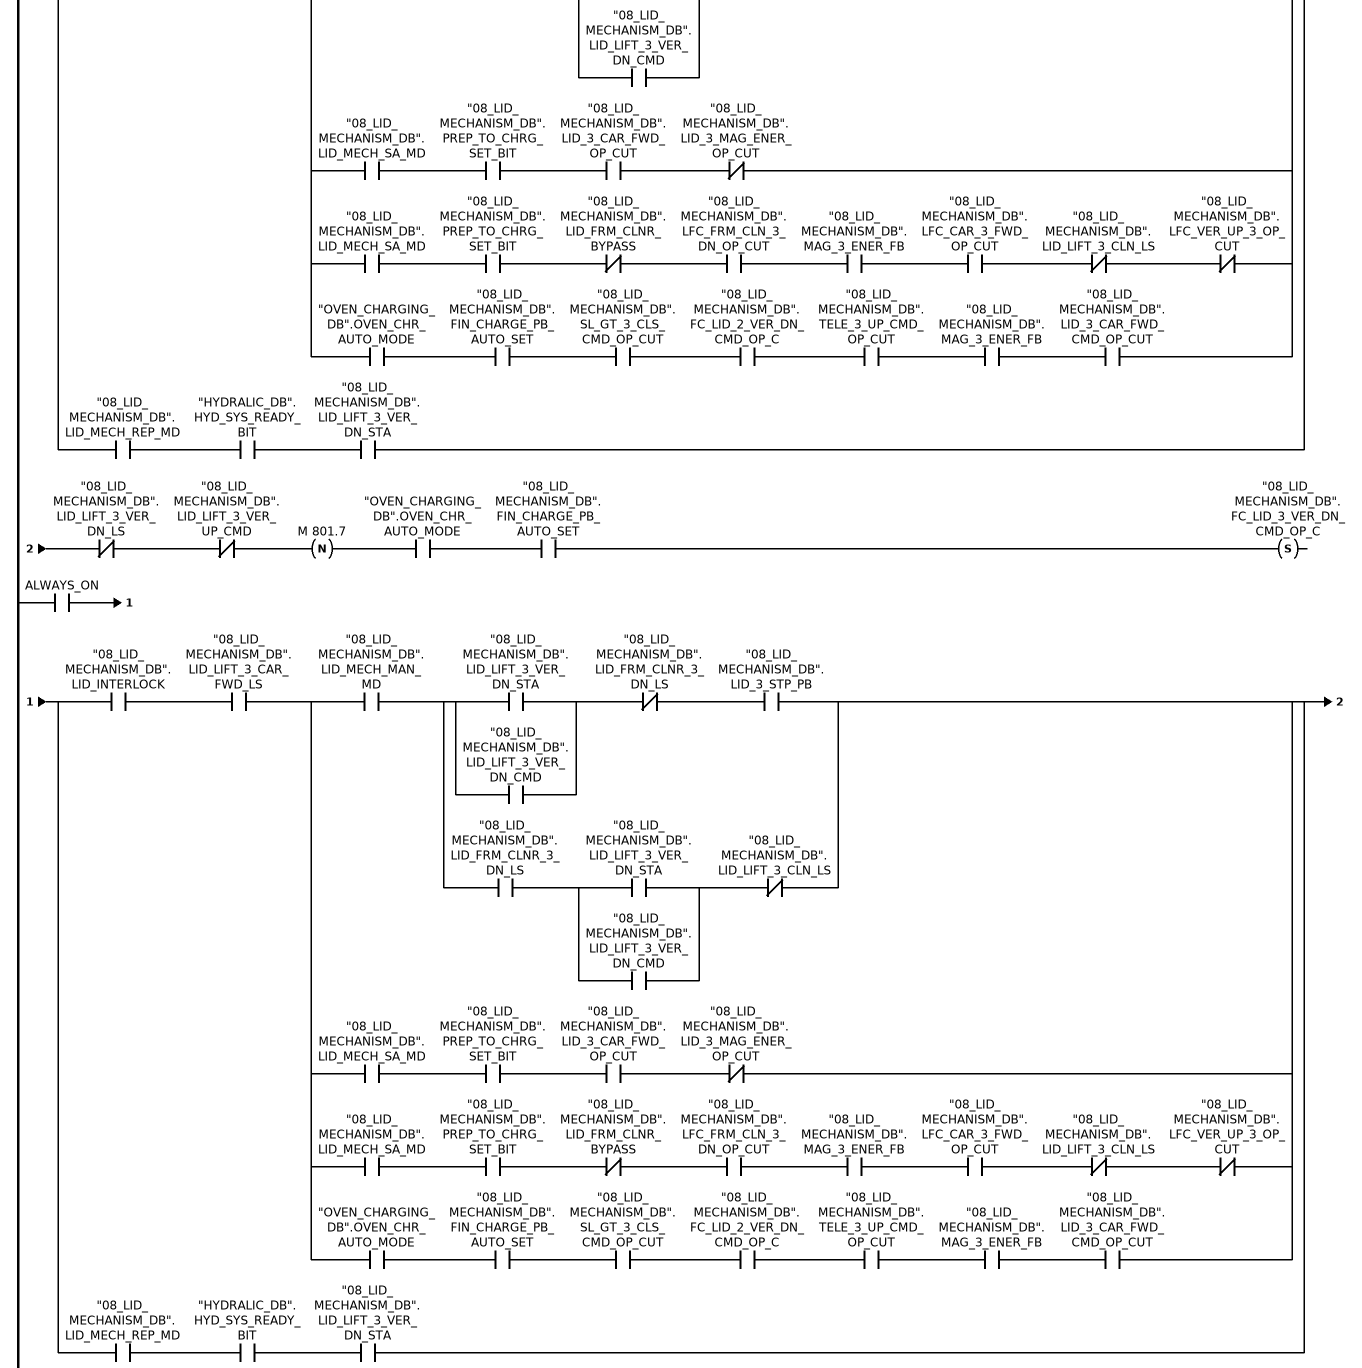
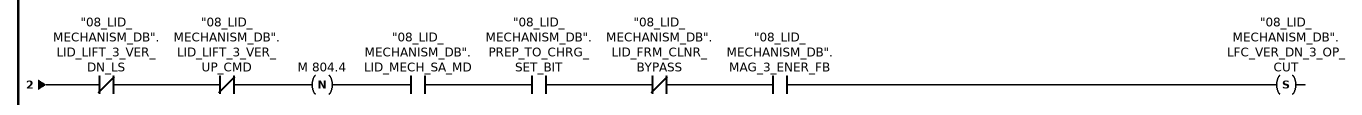
NETWORK
TITLE = LID LIFTER 3 VERTICAL DOWN COMMAND
      A     "ALWAYS_ON";
      A(;
      A     "08_LID_MECHANISM_DB".LID_INTERLOCK;
      A     "08_LID_MECHANISM_DB".LID_LIFT_3_CAR_FWD_LS;
      A(;
      A     "08_LID_MECHANISM_DB".LID_MECH_MAN_MD;
      A(;
      A(;
      O     "08_LID_MECHANISM_DB".LID_LIFT_3_VER_DN_STA;
      O     "08_LID_MECHANISM_DB".LID_LIFT_3_VER_DN_CMD;
      );
      AN    "08_LID_MECHANISM_DB".LID_FRM_CLNR_3_DN_LS;
      A     "08_LID_MECHANISM_DB".LID_3_STP_PB;
      O;
      A     "08_LID_MECHANISM_DB".LID_FRM_CLNR_3_DN_LS;
      A(;
      O     "08_LID_MECHANISM_DB".LID_LIFT_3_VER_DN_STA;
      O     "08_LID_MECHANISM_DB".LID_LIFT_3_VER_DN_CMD;
      );
      AN    "08_LID_MECHANISM_DB".LID_LIFT_3_CLN_LS;
      );
      O;
      A     "08_LID_MECHANISM_DB".LID_MECH_SA_MD;
      A     "08_LID_MECHANISM_DB".PREP_TO_CHRG_SET_BIT;
      A     "08_LID_MECHANISM_DB".LID_3_CAR_FWD_OP_CUT;
      AN    "08_LID_MECHANISM_DB".LID_3_MAG_ENER_OP_CUT;
      O;
      A     "08_LID_MECHANISM_DB".LID_MECH_SA_MD;
      A     "08_LID_MECHANISM_DB".PREP_TO_CHRG_SET_BIT;
      AN    "08_LID_MECHANISM_DB".LID_FRM_CLNR_BYPASS;
      A     "08_LID_MECHANISM_DB".LFC_FRM_CLN_3_DN_OP_CUT;
      A     "08_LID_MECHANISM_DB".MAG_3_ENER_FB;
      A     "08_LID_MECHANISM_DB".LFC_CAR_3_FWD_OP_CUT;
      AN    "08_LID_MECHANISM_DB".LID_LIFT_3_CLN_LS;
      AN    "08_LID_MECHANISM_DB".LFC_VER_UP_3_OP_CUT;
      O;
      A     "OVEN_CHARGING_DB".OVEN_CHR_AUTO_MODE;
      A     "08_LID_MECHANISM_DB".FIN_CHARGE_PB_AUTO_SET;
      A     "08_LID_MECHANISM_DB".SL_GT_3_CLS_CMD_OP_CUT;
      A     "08_LID_MECHANISM_DB".FC_LID_2_VER_DN_CMD_OP_C;
      A     "08_LID_MECHANISM_DB".TELE_3_UP_CMD_OP_CUT;
      A     "08_LID_MECHANISM_DB".MAG_3_ENER_FB;
      A     "08_LID_MECHANISM_DB".LID_3_CAR_FWD_CMD_OP_CUT;
      );
      O;
      A     "08_LID_MECHANISM_DB".LID_MECH_REP_MD;
      A     "HYDRALIC_DB".HYD_SYS_READY_BIT;
      A     "08_LID_MECHANISM_DB".LID_LIFT_3_VER_DN_STA;
      );
      AN    "08_LID_MECHANISM_DB".LID_LIFT_3_VER_DN_LS;
      AN    "08_LID_MECHANISM_DB".LID_LIFT_3_VER_UP_CMD;
      =     L 0.0;
      A     L 0.0;
      BLD   102;
      =     "08_LID_MECHANISM_DB".LID_LIFT_3_VER_DN_CMD;
      A     L 0.0;
      FP    "08_LID_MECHANISM_DB".PULSE_19;
      JNB   _005;
      L     0;
      T     "08_LID_MECHANISM_DB".LID_3_VER_DN_OP_CUT_TIME;
_005: NOP   0;
      A(;
      A     L 0.0;
      FN    M 801.7;
      );
      A     "OVEN_CHARGING_DB".OVEN_CHR_AUTO_MODE;
      A     "08_LID_MECHANISM_DB".FIN_CHARGE_PB_AUTO_SET;
      S     "08_LID_MECHANISM_DB".FC_LID_3_VER_DN_CMD_OP_C;
      A(;
      A     L 0.0;
      FN    M 804.4;
      );
      A     "08_LID_MECHANISM_DB".LID_MECH_SA_MD;
      A     "08_LID_MECHANISM_DB".PREP_TO_CHRG_SET_BIT;
      AN    "08_LID_MECHANISM_DB".LID_FRM_CLNR_BYPASS;
      A     "08_LID_MECHANISM_DB".MAG_3_ENER_FB;
      S     "08_LID_MECHANISM_DB".LFC_VER_DN_3_OP_CUT;
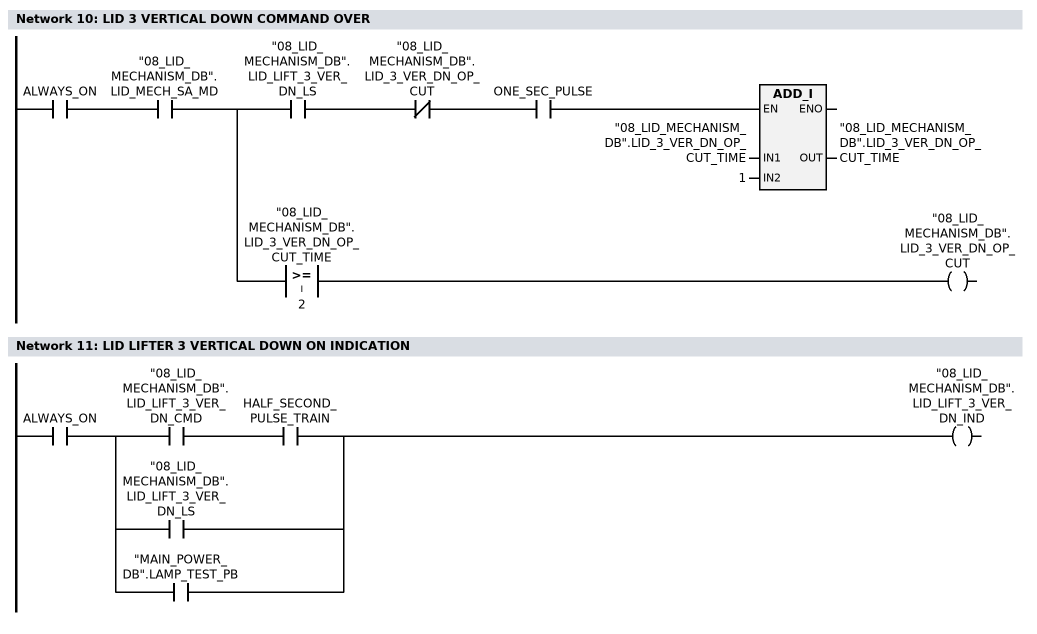
NETWORK
TITLE = LID 3 VERTICAL DOWN COMMAND OVER
      A     "ALWAYS_ON";
      A     "08_LID_MECHANISM_DB".LID_MECH_SA_MD;
      =     L 0.0;
      A     L 0.0;
      A     "08_LID_MECHANISM_DB".LID_LIFT_3_VER_DN_LS;
      AN    "08_LID_MECHANISM_DB".LID_3_VER_DN_OP_CUT;
      A     "ONE_SEC_PULSE";
      JNB   _006;
      L     "08_LID_MECHANISM_DB".LID_3_VER_DN_OP_CUT_TIME;
      L     1;
      +I;
      T     "08_LID_MECHANISM_DB".LID_3_VER_DN_OP_CUT_TIME;
_006: NOP   0;
      A     L 0.0;
      A(;
      L     "08_LID_MECHANISM_DB".LID_3_VER_DN_OP_CUT_TIME;
      L     2;
      >=I;
      );
      =     "08_LID_MECHANISM_DB".LID_3_VER_DN_OP_CUT;
NETWORK
TITLE = LID LIFTER 3 VERTICAL DOWN ON INDICATION
      A     "ALWAYS_ON";
      A(;
      A     "08_LID_MECHANISM_DB".LID_LIFT_3_VER_DN_CMD;
      A     "HALF_SECOND_PULSE_TRAIN";
      O     "08_LID_MECHANISM_DB".LID_LIFT_3_VER_DN_LS;
      O     "MAIN_POWER_DB".LAMP_TEST_PB;
      );
      =     "08_LID_MECHANISM_DB".LID_LIFT_3_VER_DN_IND;
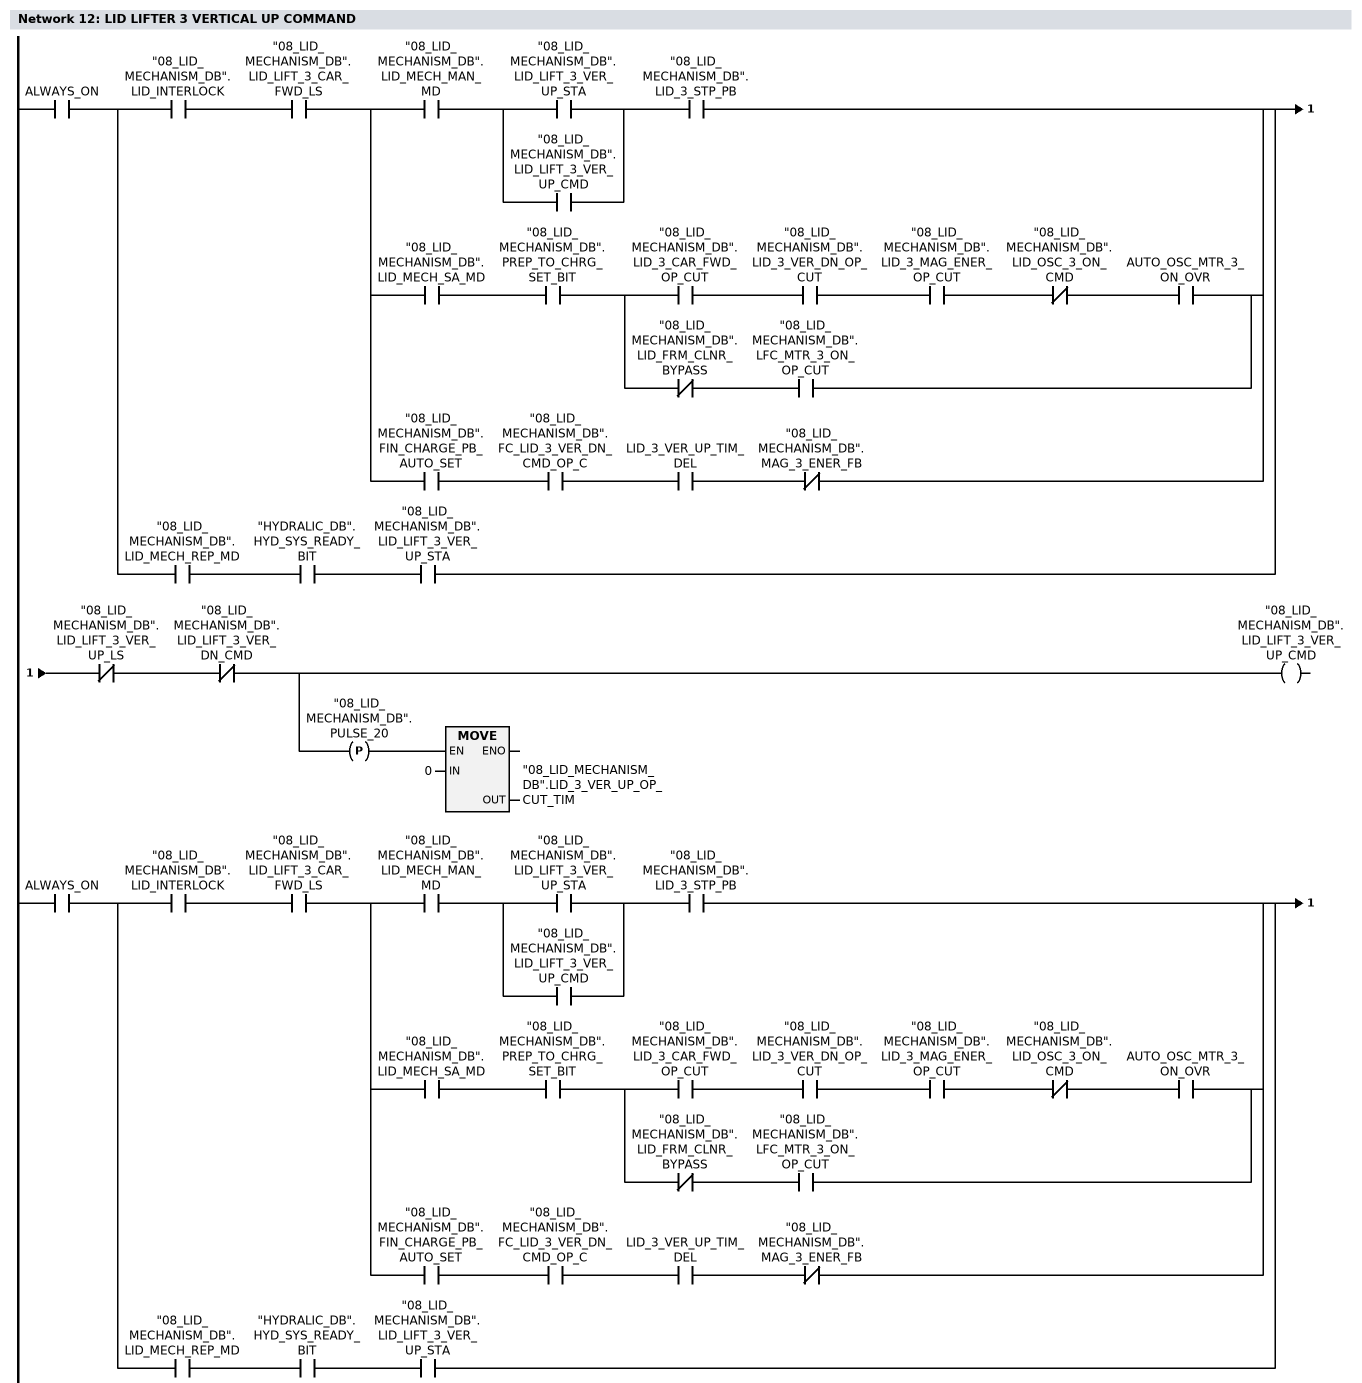
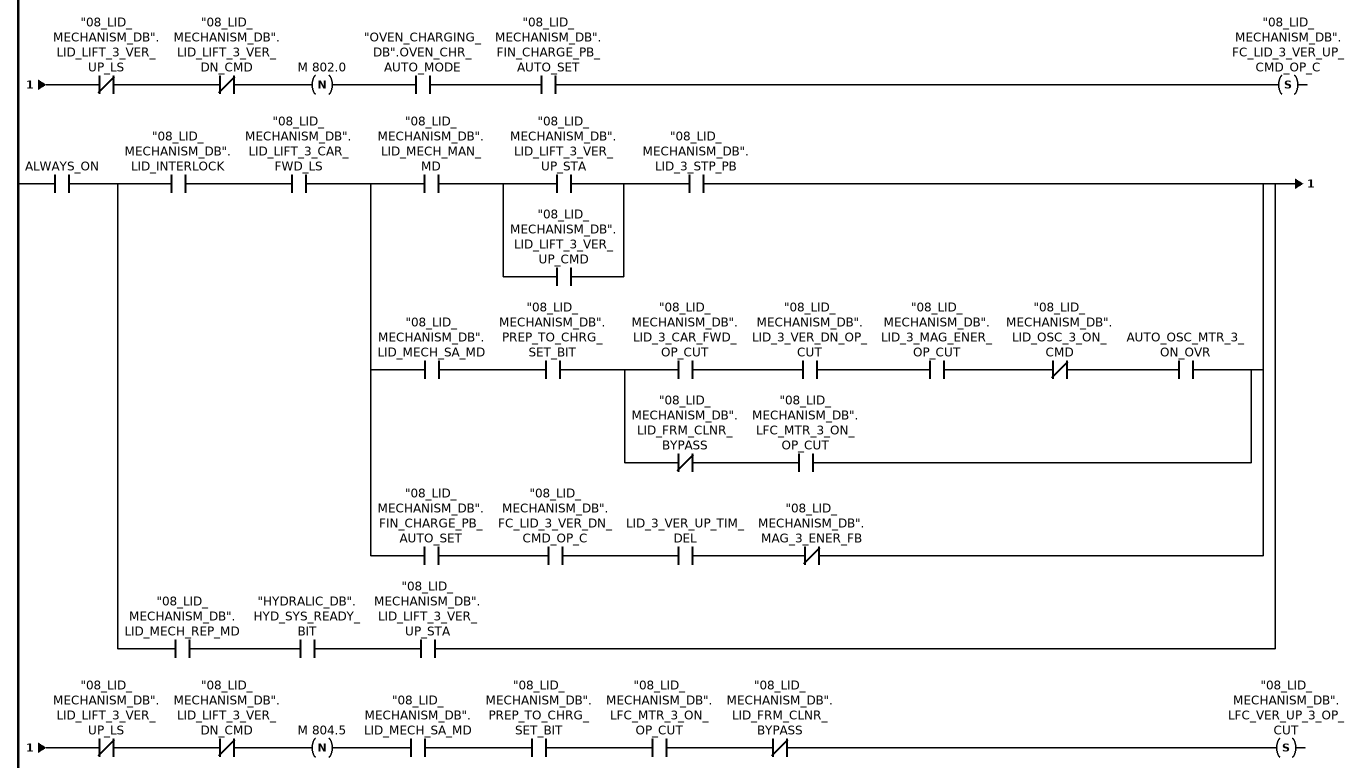
NETWORK
TITLE = LID LIFTER 3 VERTICAL UP COMMAND
      A     "ALWAYS_ON";
      A(;
      A     "08_LID_MECHANISM_DB".LID_INTERLOCK;
      A     "08_LID_MECHANISM_DB".LID_LIFT_3_CAR_FWD_LS;
      A(;
      A     "08_LID_MECHANISM_DB".LID_MECH_MAN_MD;
      A(;
      O     "08_LID_MECHANISM_DB".LID_LIFT_3_VER_UP_STA;
      O     "08_LID_MECHANISM_DB".LID_LIFT_3_VER_UP_CMD;
      );
      A     "08_LID_MECHANISM_DB".LID_3_STP_PB;
      O;
      A     "08_LID_MECHANISM_DB".LID_MECH_SA_MD;
      A     "08_LID_MECHANISM_DB".PREP_TO_CHRG_SET_BIT;
      A(;
      A     "08_LID_MECHANISM_DB".LID_3_CAR_FWD_OP_CUT;
      A     "08_LID_MECHANISM_DB".LID_3_VER_DN_OP_CUT;
      A     "08_LID_MECHANISM_DB".LID_3_MAG_ENER_OP_CUT;
      AN    "08_LID_MECHANISM_DB".LID_OSC_3_ON_CMD;
      A     "AUTO_OSC_MTR_3_ON_OVR";
      O;
      AN    "08_LID_MECHANISM_DB".LID_FRM_CLNR_BYPASS;
      A     "08_LID_MECHANISM_DB".LFC_MTR_3_ON_OP_CUT;
      );
      O;
      A     "08_LID_MECHANISM_DB".FIN_CHARGE_PB_AUTO_SET;
      A     "08_LID_MECHANISM_DB".FC_LID_3_VER_DN_CMD_OP_C;
      A     "LID_3_VER_UP_TIM_DEL";
      AN    "08_LID_MECHANISM_DB".MAG_3_ENER_FB;
      );
      O;
      A     "08_LID_MECHANISM_DB".LID_MECH_REP_MD;
      A     "HYDRALIC_DB".HYD_SYS_READY_BIT;
      A     "08_LID_MECHANISM_DB".LID_LIFT_3_VER_UP_STA;
      );
      AN    "08_LID_MECHANISM_DB".LID_LIFT_3_VER_UP_LS;
      AN    "08_LID_MECHANISM_DB".LID_LIFT_3_VER_DN_CMD;
      =     L 0.0;
      A     L 0.0;
      BLD   102;
      =     "08_LID_MECHANISM_DB".LID_LIFT_3_VER_UP_CMD;
      A     L 0.0;
      FP    "08_LID_MECHANISM_DB".PULSE_20;
      JNB   _007;
      L     0;
      T     "08_LID_MECHANISM_DB".LID_3_VER_UP_OP_CUT_TIM;
_007: NOP   0;
      A(;
      A     L 0.0;
      FN    M 802.0;
      );
      A     "OVEN_CHARGING_DB".OVEN_CHR_AUTO_MODE;
      A     "08_LID_MECHANISM_DB".FIN_CHARGE_PB_AUTO_SET;
      S     "08_LID_MECHANISM_DB".FC_LID_3_VER_UP_CMD_OP_C;
      A(;
      A     L 0.0;
      FN    M 804.5;
      );
      A     "08_LID_MECHANISM_DB".LID_MECH_SA_MD;
      A     "08_LID_MECHANISM_DB".PREP_TO_CHRG_SET_BIT;
      A     "08_LID_MECHANISM_DB".LFC_MTR_3_ON_OP_CUT;
      AN    "08_LID_MECHANISM_DB".LID_FRM_CLNR_BYPASS;
      S     "08_LID_MECHANISM_DB".LFC_VER_UP_3_OP_CUT;
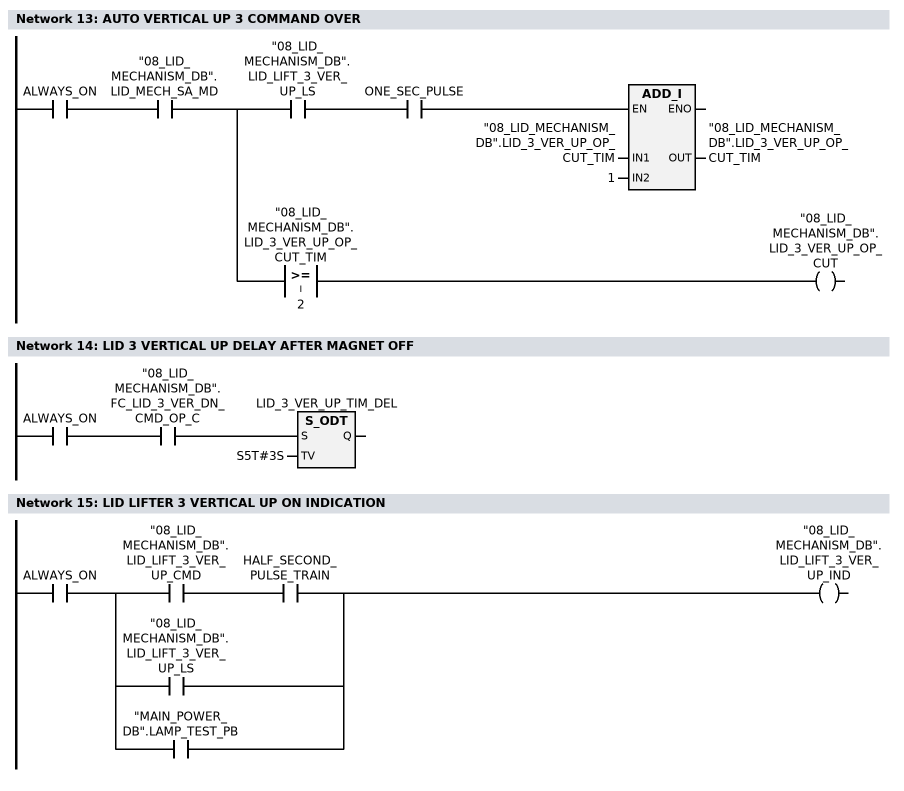
NETWORK
TITLE = AUTO VERTICAL UP 3 COMMAND OVER
      A     "ALWAYS_ON";
      A     "08_LID_MECHANISM_DB".LID_MECH_SA_MD;
      =     L 0.0;
      A     L 0.0;
      A     "08_LID_MECHANISM_DB".LID_LIFT_3_VER_UP_LS;
      A     "ONE_SEC_PULSE";
      JNB   _008;
      L     "08_LID_MECHANISM_DB".LID_3_VER_UP_OP_CUT_TIM;
      L     1;
      +I;
      T     "08_LID_MECHANISM_DB".LID_3_VER_UP_OP_CUT_TIM;
_008: NOP   0;
      A     L 0.0;
      A(;
      L     "08_LID_MECHANISM_DB".LID_3_VER_UP_OP_CUT_TIM;
      L     2;
      >=I;
      );
      =     "08_LID_MECHANISM_DB".LID_3_VER_UP_OP_CUT;
NETWORK
TITLE = LID 3 VERTICAL UP DELAY AFTER MAGNET OFF
      A     "ALWAYS_ON";
      A     "08_LID_MECHANISM_DB".FC_LID_3_VER_DN_CMD_OP_C;
      L     S5T#3S;
      SD    "LID_3_VER_UP_TIM_DEL";
      NOP   0;
      NOP   0;
      NOP   0;
      NOP   0;
NETWORK
TITLE = LID LIFTER 3 VERTICAL UP ON INDICATION
      A     "ALWAYS_ON";
      A(;
      A     "08_LID_MECHANISM_DB".LID_LIFT_3_VER_UP_CMD;
      A     "HALF_SECOND_PULSE_TRAIN";
      O     "08_LID_MECHANISM_DB".LID_LIFT_3_VER_UP_LS;
      O     "MAIN_POWER_DB".LAMP_TEST_PB;
      );
      =     "08_LID_MECHANISM_DB".LID_LIFT_3_VER_UP_IND;
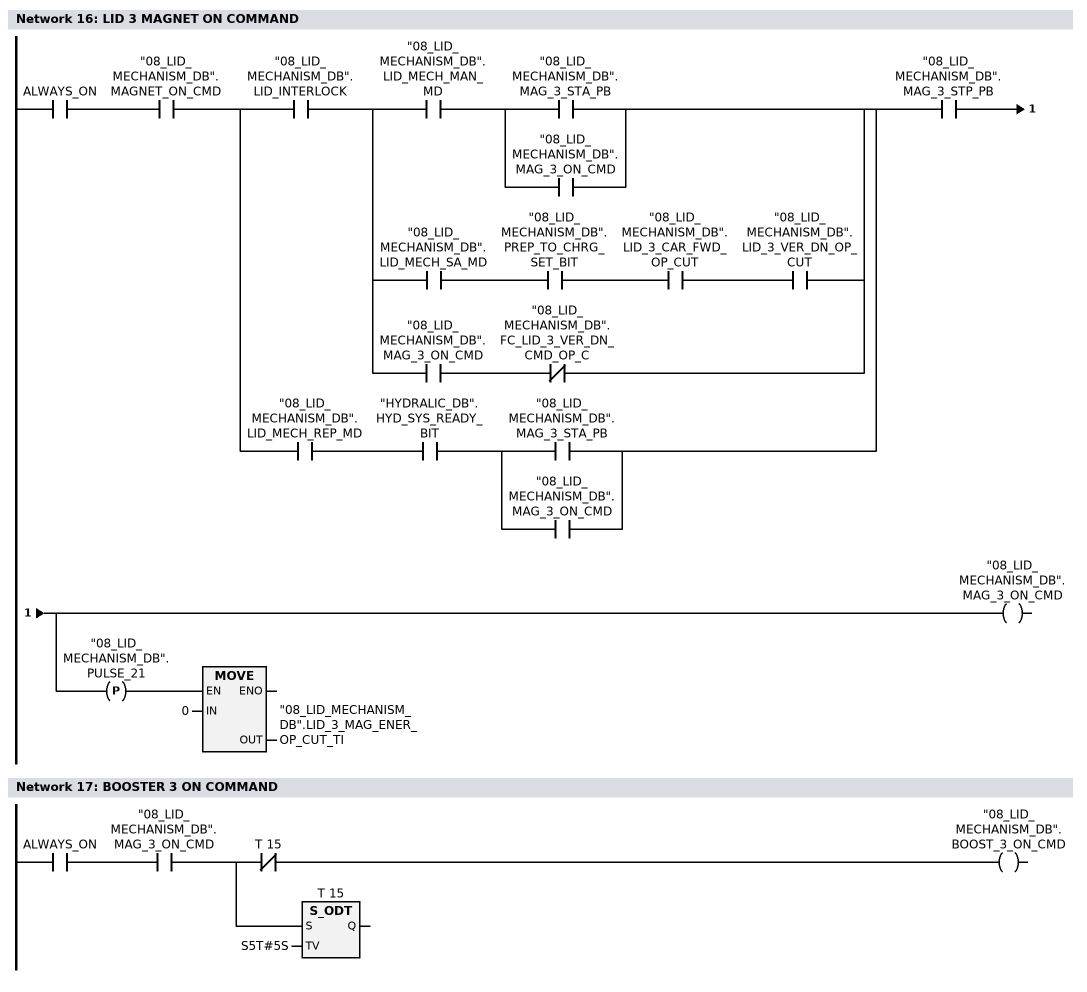
NETWORK
TITLE = LID 3 MAGNET ON COMMAND
      A     "ALWAYS_ON";
      A     "08_LID_MECHANISM_DB".MAGNET_ON_CMD;
      A(;
      A     "08_LID_MECHANISM_DB".LID_INTERLOCK;
      A(;
      A     "08_LID_MECHANISM_DB".LID_MECH_MAN_MD;
      A(;
      O     "08_LID_MECHANISM_DB".MAG_3_STA_PB;
      O     "08_LID_MECHANISM_DB".MAG_3_ON_CMD;
      );
      O;
      A     "08_LID_MECHANISM_DB".LID_MECH_SA_MD;
      A     "08_LID_MECHANISM_DB".PREP_TO_CHRG_SET_BIT;
      A     "08_LID_MECHANISM_DB".LID_3_CAR_FWD_OP_CUT;
      A     "08_LID_MECHANISM_DB".LID_3_VER_DN_OP_CUT;
      O;
      A     "08_LID_MECHANISM_DB".MAG_3_ON_CMD;
      AN    "08_LID_MECHANISM_DB".FC_LID_3_VER_DN_CMD_OP_C;
      );
      O;
      A     "08_LID_MECHANISM_DB".LID_MECH_REP_MD;
      A     "HYDRALIC_DB".HYD_SYS_READY_BIT;
      A(;
      O     "08_LID_MECHANISM_DB".MAG_3_STA_PB;
      O     "08_LID_MECHANISM_DB".MAG_3_ON_CMD;
      );
      );
      A     "08_LID_MECHANISM_DB".MAG_3_STP_PB;
      =     L 0.0;
      A     L 0.0;
      BLD   102;
      =     "08_LID_MECHANISM_DB".MAG_3_ON_CMD;
      A     L 0.0;
      FP    "08_LID_MECHANISM_DB".PULSE_21;
      JNB   _009;
      L     0;
      T     "08_LID_MECHANISM_DB".LID_3_MAG_ENER_OP_CUT_TI;
_009: NOP   0;
NETWORK
TITLE = BOOSTER 3 ON COMMAND
      A     "ALWAYS_ON";
      A     "08_LID_MECHANISM_DB".MAG_3_ON_CMD;
      =     L 0.0;
      A     L 0.0;
      AN    T 15;
      =     "08_LID_MECHANISM_DB".BOOST_3_ON_CMD;
      A     L 0.0;
      L     S5T#5S;
      SD    T 15;
      NOP   0;
      NOP   0;
      NOP   0;
      NOP   0;
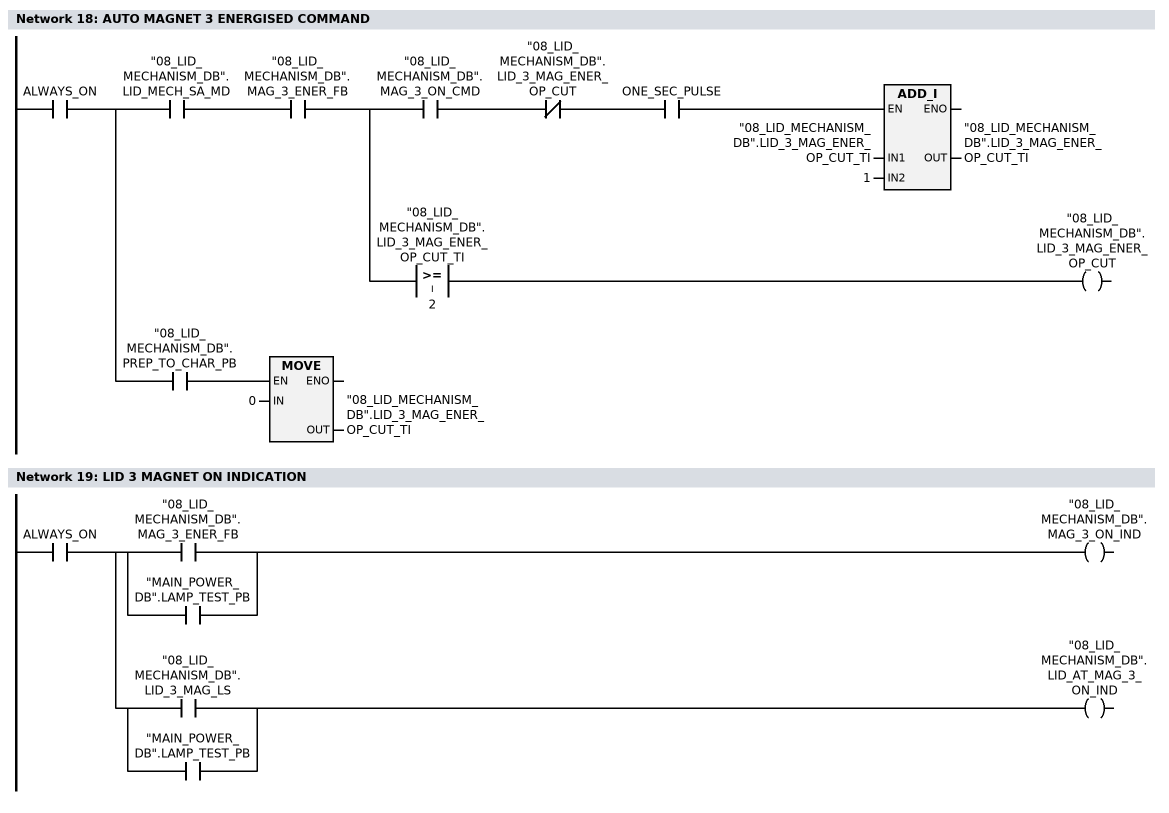
NETWORK
TITLE = AUTO MAGNET 3 ENERGISED COMMAND
      A     "ALWAYS_ON";
      =     L 0.0;
      A     L 0.0;
      A     "08_LID_MECHANISM_DB".LID_MECH_SA_MD;
      A     "08_LID_MECHANISM_DB".MAG_3_ENER_FB;
      =     L 0.1;
      A     L 0.1;
      A     "08_LID_MECHANISM_DB".MAG_3_ON_CMD;
      AN    "08_LID_MECHANISM_DB".LID_3_MAG_ENER_OP_CUT;
      A     "ONE_SEC_PULSE";
      JNB   _00a;
      L     "08_LID_MECHANISM_DB".LID_3_MAG_ENER_OP_CUT_TI;
      L     1;
      +I;
      T     "08_LID_MECHANISM_DB".LID_3_MAG_ENER_OP_CUT_TI;
_00a: NOP   0;
      A     L 0.1;
      A(;
      L     "08_LID_MECHANISM_DB".LID_3_MAG_ENER_OP_CUT_TI;
      L     2;
      >=I;
      );
      =     "08_LID_MECHANISM_DB".LID_3_MAG_ENER_OP_CUT;
      A     L 0.0;
      A     "08_LID_MECHANISM_DB".PREP_TO_CHAR_PB;
      JNB   _00b;
      L     0;
      T     "08_LID_MECHANISM_DB".LID_3_MAG_ENER_OP_CUT_TI;
_00b: NOP   0;
NETWORK
TITLE = LID 3 MAGNET ON INDICATION
      A     "ALWAYS_ON";
      =     L 0.0;
      A     L 0.0;
      A(;
      O     "08_LID_MECHANISM_DB".MAG_3_ENER_FB;
      O     "MAIN_POWER_DB".LAMP_TEST_PB;
      );
      =     "08_LID_MECHANISM_DB".MAG_3_ON_IND;
      A     L 0.0;
      A(;
      O     "08_LID_MECHANISM_DB".LID_3_MAG_LS;
      O     "MAIN_POWER_DB".LAMP_TEST_PB;
      );
      =     "08_LID_MECHANISM_DB".LID_AT_MAG_3_ON_IND;
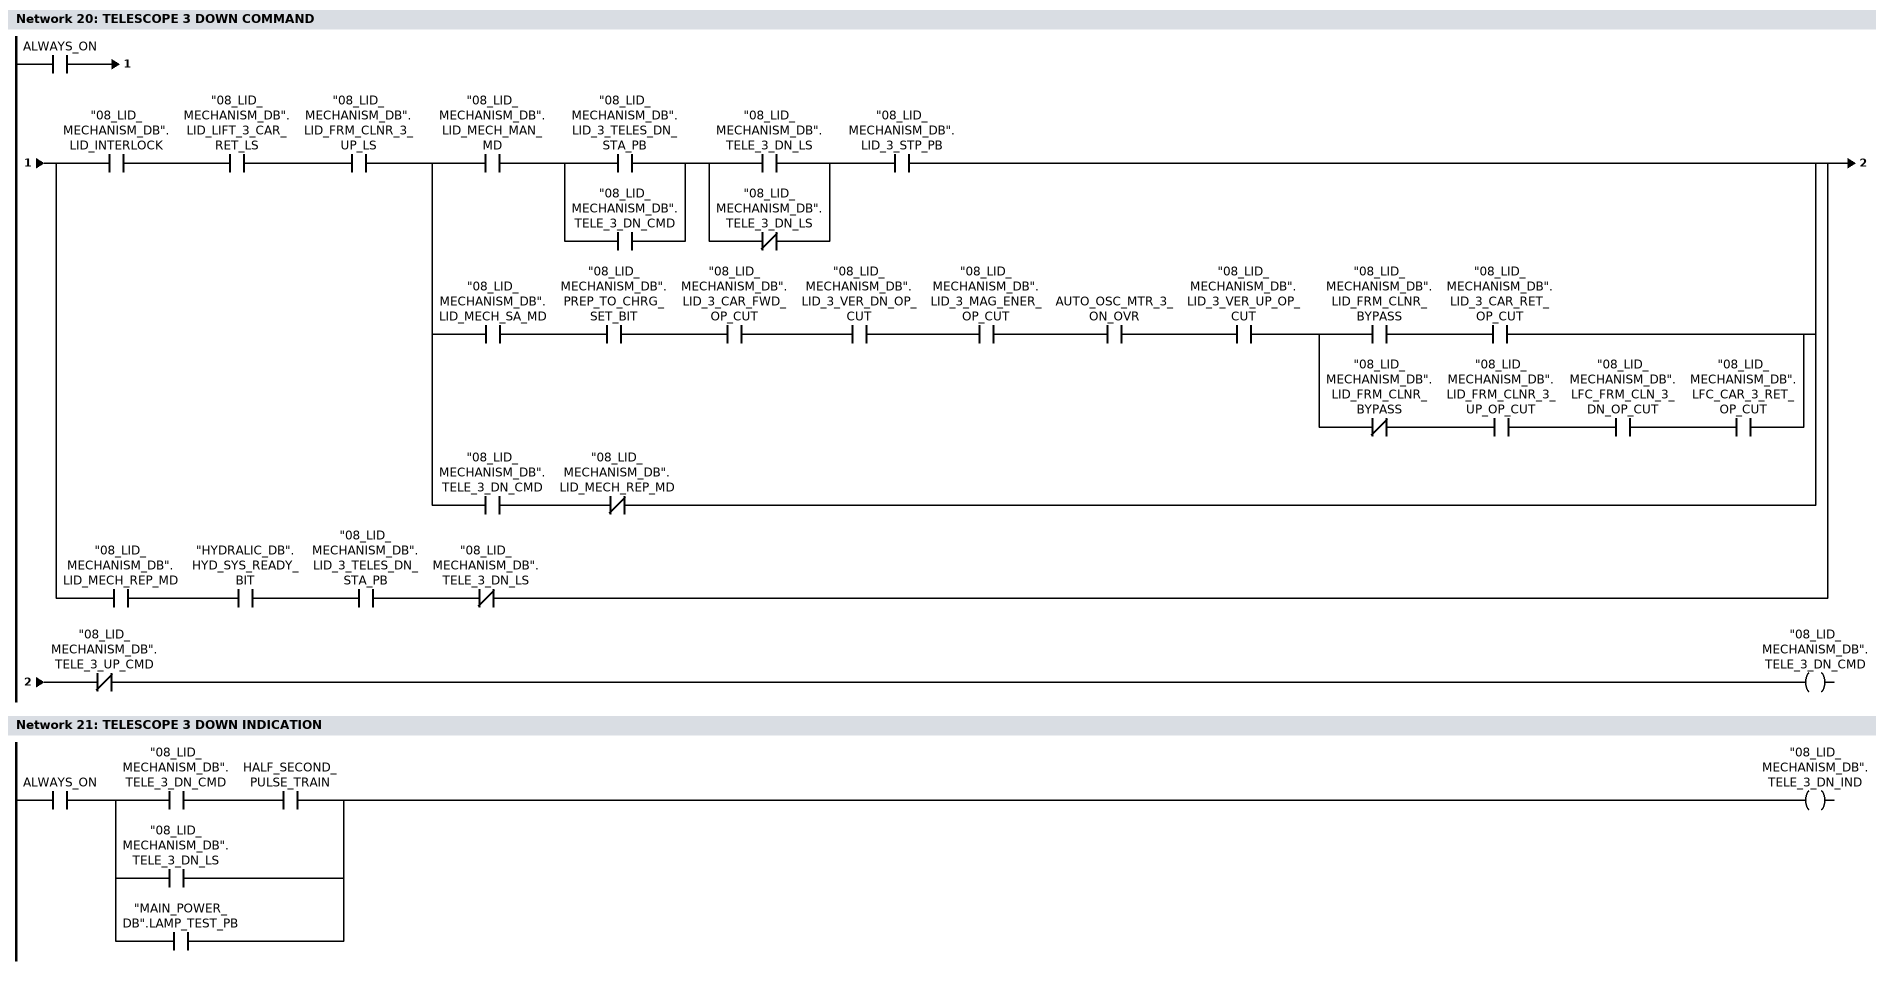
NETWORK
TITLE = TELESCOPE 3 DOWN COMMAND
      A     "ALWAYS_ON";
      A(;
      A     "08_LID_MECHANISM_DB".LID_INTERLOCK;
      A     "08_LID_MECHANISM_DB".LID_LIFT_3_CAR_RET_LS;
      A     "08_LID_MECHANISM_DB".LID_FRM_CLNR_3_UP_LS;
      A(;
      A     "08_LID_MECHANISM_DB".LID_MECH_MAN_MD;
      A(;
      O     "08_LID_MECHANISM_DB".LID_3_TELES_DN_STA_PB;
      O     "08_LID_MECHANISM_DB".TELE_3_DN_CMD;
      );
      A(;
      O     "08_LID_MECHANISM_DB".TELE_3_DN_LS;
      ON    "08_LID_MECHANISM_DB".TELE_3_DN_LS;
      );
      A     "08_LID_MECHANISM_DB".LID_3_STP_PB;
      O;
      A     "08_LID_MECHANISM_DB".LID_MECH_SA_MD;
      A     "08_LID_MECHANISM_DB".PREP_TO_CHRG_SET_BIT;
      A     "08_LID_MECHANISM_DB".LID_3_CAR_FWD_OP_CUT;
      A     "08_LID_MECHANISM_DB".LID_3_VER_DN_OP_CUT;
      A     "08_LID_MECHANISM_DB".LID_3_MAG_ENER_OP_CUT;
      A     "AUTO_OSC_MTR_3_ON_OVR";
      A     "08_LID_MECHANISM_DB".LID_3_VER_UP_OP_CUT;
      A(;
      A     "08_LID_MECHANISM_DB".LID_FRM_CLNR_BYPASS;
      A     "08_LID_MECHANISM_DB".LID_3_CAR_RET_OP_CUT;
      O;
      AN    "08_LID_MECHANISM_DB".LID_FRM_CLNR_BYPASS;
      A     "08_LID_MECHANISM_DB".LID_FRM_CLNR_3_UP_OP_CUT;
      A     "08_LID_MECHANISM_DB".LFC_FRM_CLN_3_DN_OP_CUT;
      A     "08_LID_MECHANISM_DB".LFC_CAR_3_RET_OP_CUT;
      );
      O;
      A     "08_LID_MECHANISM_DB".TELE_3_DN_CMD;
      AN    "08_LID_MECHANISM_DB".LID_MECH_REP_MD;
      );
      O;
      A     "08_LID_MECHANISM_DB".LID_MECH_REP_MD;
      A     "HYDRALIC_DB".HYD_SYS_READY_BIT;
      A     "08_LID_MECHANISM_DB".LID_3_TELES_DN_STA_PB;
      AN    "08_LID_MECHANISM_DB".TELE_3_DN_LS;
      );
      AN    "08_LID_MECHANISM_DB".TELE_3_UP_CMD;
      =     "08_LID_MECHANISM_DB".TELE_3_DN_CMD;
NETWORK
TITLE = TELESCOPE 3 DOWN INDICATION
      A     "ALWAYS_ON";
      A(;
      A     "08_LID_MECHANISM_DB".TELE_3_DN_CMD;
      A     "HALF_SECOND_PULSE_TRAIN";
      O     "08_LID_MECHANISM_DB".TELE_3_DN_LS;
      O     "MAIN_POWER_DB".LAMP_TEST_PB;
      );
      =     "08_LID_MECHANISM_DB".TELE_3_DN_IND;
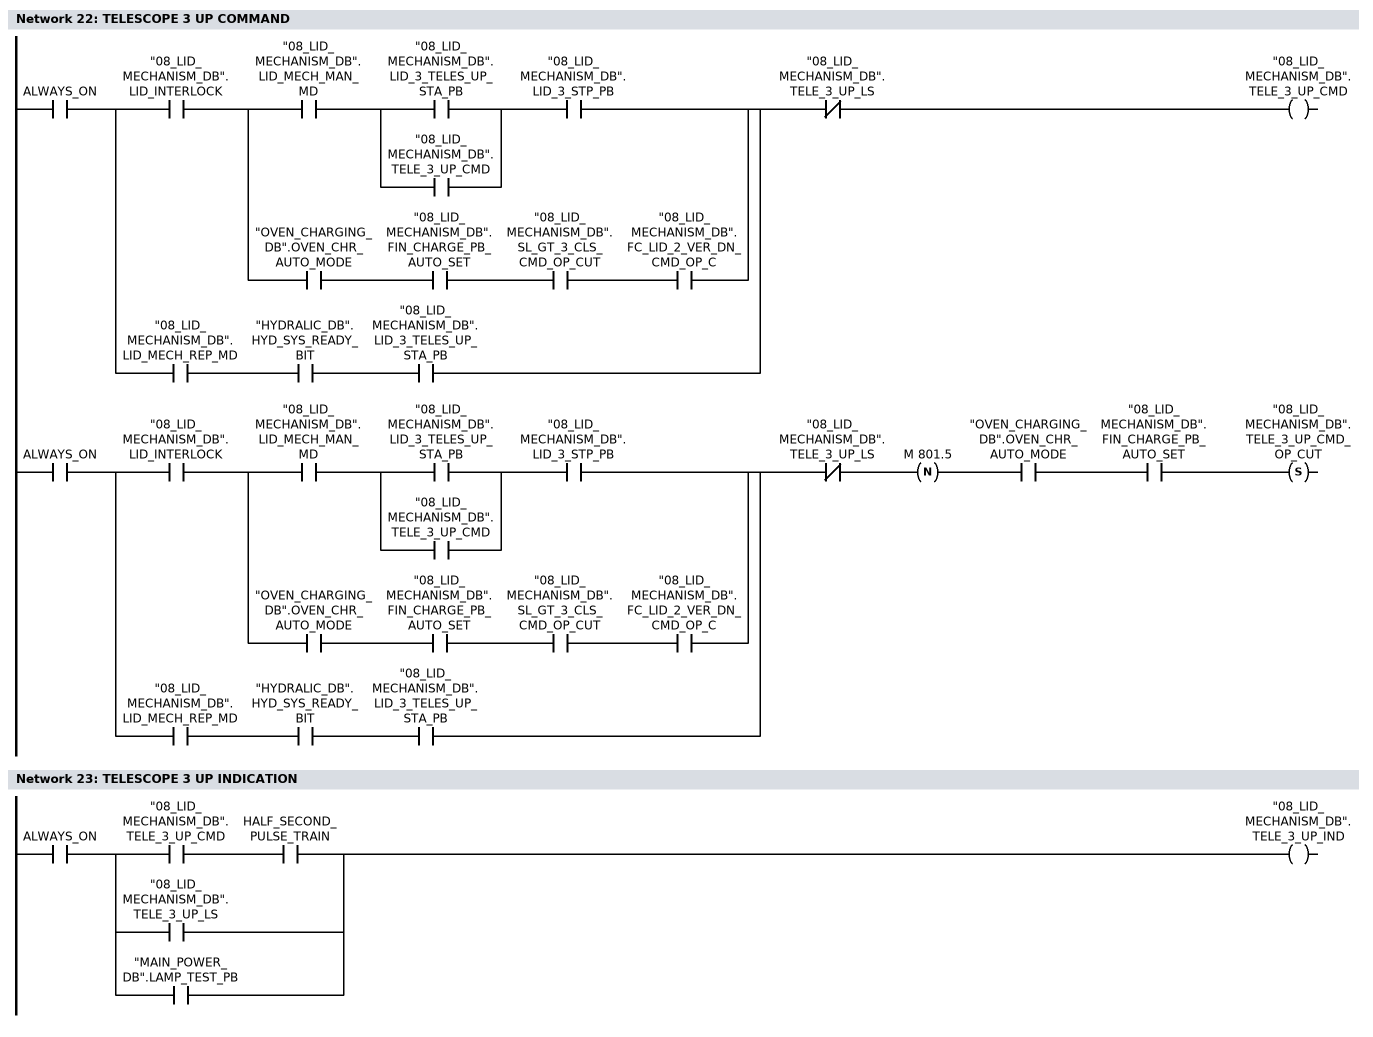
NETWORK
TITLE = TELESCOPE 3 UP COMMAND
      A     "ALWAYS_ON";
      A(;
      A     "08_LID_MECHANISM_DB".LID_INTERLOCK;
      A(;
      A     "08_LID_MECHANISM_DB".LID_MECH_MAN_MD;
      A(;
      O     "08_LID_MECHANISM_DB".LID_3_TELES_UP_STA_PB;
      O     "08_LID_MECHANISM_DB".TELE_3_UP_CMD;
      );
      A     "08_LID_MECHANISM_DB".LID_3_STP_PB;
      O;
      A     "OVEN_CHARGING_DB".OVEN_CHR_AUTO_MODE;
      A     "08_LID_MECHANISM_DB".FIN_CHARGE_PB_AUTO_SET;
      A     "08_LID_MECHANISM_DB".SL_GT_3_CLS_CMD_OP_CUT;
      A     "08_LID_MECHANISM_DB".FC_LID_2_VER_DN_CMD_OP_C;
      );
      O;
      A     "08_LID_MECHANISM_DB".LID_MECH_REP_MD;
      A     "HYDRALIC_DB".HYD_SYS_READY_BIT;
      A     "08_LID_MECHANISM_DB".LID_3_TELES_UP_STA_PB;
      );
      AN    "08_LID_MECHANISM_DB".TELE_3_UP_LS;
      =     L 0.0;
      A     L 0.0;
      BLD   102;
      =     "08_LID_MECHANISM_DB".TELE_3_UP_CMD;
      A(;
      A     L 0.0;
      FN    M 801.5;
      );
      A     "OVEN_CHARGING_DB".OVEN_CHR_AUTO_MODE;
      A     "08_LID_MECHANISM_DB".FIN_CHARGE_PB_AUTO_SET;
      S     "08_LID_MECHANISM_DB".TELE_3_UP_CMD_OP_CUT;
NETWORK
TITLE = TELESCOPE 3 UP INDICATION
      A     "ALWAYS_ON";
      A(;
      A     "08_LID_MECHANISM_DB".TELE_3_UP_CMD;
      A     "HALF_SECOND_PULSE_TRAIN";
      O     "08_LID_MECHANISM_DB".TELE_3_UP_LS;
      O     "MAIN_POWER_DB".LAMP_TEST_PB;
      );
      =     "08_LID_MECHANISM_DB".TELE_3_UP_IND;
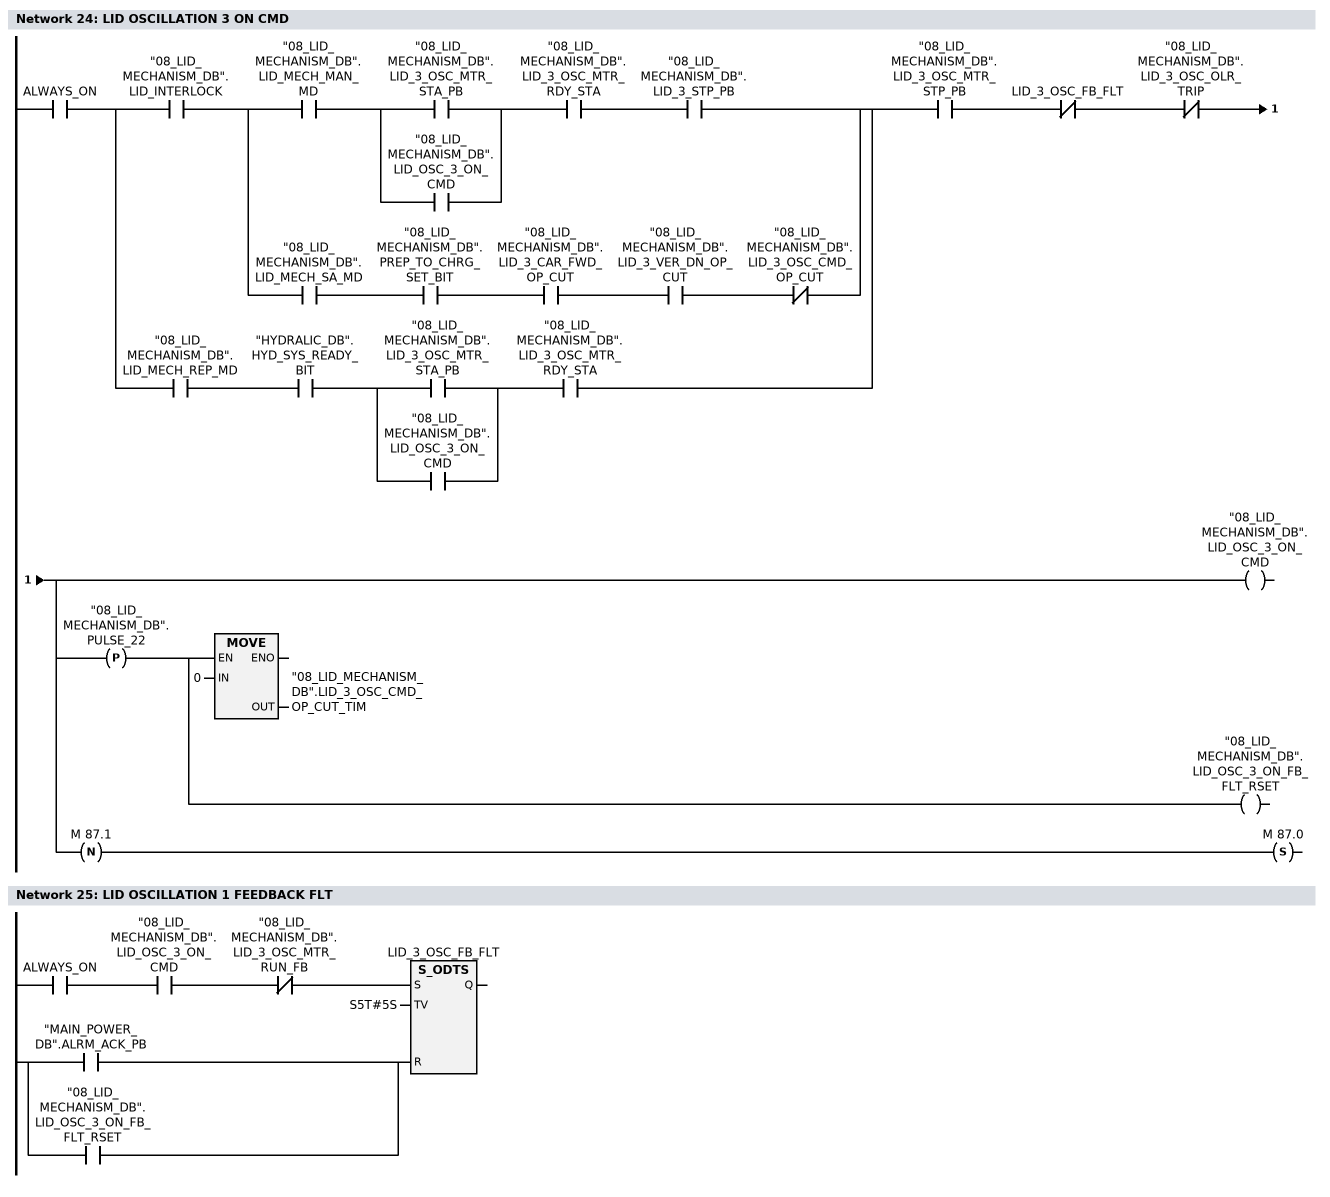
NETWORK
TITLE = LID OSCILLATION 3 ON CMD
      A     "ALWAYS_ON";
      A(;
      A     "08_LID_MECHANISM_DB".LID_INTERLOCK;
      A(;
      A     "08_LID_MECHANISM_DB".LID_MECH_MAN_MD;
      A(;
      O     "08_LID_MECHANISM_DB".LID_3_OSC_MTR_STA_PB;
      O     "08_LID_MECHANISM_DB".LID_OSC_3_ON_CMD;
      );
      A     "08_LID_MECHANISM_DB".LID_3_OSC_MTR_RDY_STA;
      A     "08_LID_MECHANISM_DB".LID_3_STP_PB;
      O;
      A     "08_LID_MECHANISM_DB".LID_MECH_SA_MD;
      A     "08_LID_MECHANISM_DB".PREP_TO_CHRG_SET_BIT;
      A     "08_LID_MECHANISM_DB".LID_3_CAR_FWD_OP_CUT;
      A     "08_LID_MECHANISM_DB".LID_3_VER_DN_OP_CUT;
      AN    "08_LID_MECHANISM_DB".LID_3_OSC_CMD_OP_CUT;
      );
      O;
      A     "08_LID_MECHANISM_DB".LID_MECH_REP_MD;
      A     "HYDRALIC_DB".HYD_SYS_READY_BIT;
      A(;
      O     "08_LID_MECHANISM_DB".LID_3_OSC_MTR_STA_PB;
      O     "08_LID_MECHANISM_DB".LID_OSC_3_ON_CMD;
      );
      A     "08_LID_MECHANISM_DB".LID_3_OSC_MTR_RDY_STA;
      );
      A     "08_LID_MECHANISM_DB".LID_3_OSC_MTR_STP_PB;
      AN    "LID_3_OSC_FB_FLT";
      AN    "08_LID_MECHANISM_DB".LID_3_OSC_OLR_TRIP;
      =     L 0.0;
      A     L 0.0;
      BLD   102;
      =     "08_LID_MECHANISM_DB".LID_OSC_3_ON_CMD;
      A     L 0.0;
      FP    "08_LID_MECHANISM_DB".PULSE_22;
      =     L 0.1;
      A     L 0.1;
      JNB   _00c;
      L     0;
      T     "08_LID_MECHANISM_DB".LID_3_OSC_CMD_OP_CUT_TIM;
_00c: NOP   0;
      A     L 0.1;
      BLD   102;
      =     "08_LID_MECHANISM_DB".LID_OSC_3_ON_FB_FLT_RSET;
      A     L 0.0;
      FN    M 87.1;
      S     M 87.0;
NETWORK
TITLE = LID OSCILLATION 1 FEEDBACK FLT
      A     "ALWAYS_ON";
      A     "08_LID_MECHANISM_DB".LID_OSC_3_ON_CMD;
      AN    "08_LID_MECHANISM_DB".LID_3_OSC_MTR_RUN_FB;
      L     S5T#5S;
      SS    "LID_3_OSC_FB_FLT";
      A(;
      O     "MAIN_POWER_DB".ALRM_ACK_PB;
      O     "08_LID_MECHANISM_DB".LID_OSC_3_ON_FB_FLT_RSET;
      );
      R     "LID_3_OSC_FB_FLT";
      NOP   0;
      NOP   0;
      NOP   0;
